    20: (* Transition Delay After Last Bin (Bin 10) Closes *)
        Active_Material_ID := 0;
        Active_Bin_ID := 0;
        Active_Target_Weight := 0.0;
        Status_Message := 'Settling Last Bin';
        Transition_Timer(IN := TRUE, PT := Step_Delay_Time);
        IF Transition_Timer.Q THEN
            Transition_Timer(IN := FALSE);
            Step := 30; // Go to post-discharge wait step (State 30)
        END_IF;

    30: (* Wait 2 Seconds After Closing the Last Bin *)
        Active_Material_ID := 0;
        Active_Bin_ID := 0;
        Active_Target_Weight := 0.0;
        Status_Message := 'Settling Delay';
        Completion_Timer(IN := TRUE, PT := Post_Complete_Delay);
        IF Completion_Timer.Q THEN
            Completion_Timer(IN := FALSE);
            Step := 40; // Proceed to reset last weight (State 40)
        END_IF;
        
    40: (* Reset bin_last_weight to 0 & Complete *)
        Active_Material_ID := 0;
        Active_Bin_ID := 0;
        Active_Target_Weight := 0.0;
        Status_Message := 'Sequence Completed';
        bin_last_weight := 0.0;
        Sequence_Complete := TRUE;
        
        IF NOT Start_Button THEN
            Step := 0;
            Sequence_Complete := FALSE;
            (* Reset all actual weights at completion once start is released *)
            FOR i := 1 TO 10 DO
                Actual_Weights[i] := 0.0;
            END_FOR;
        END_IF;
        
    99: (* Error Abort state *)
        FOR i := 1 TO 10 DO 
            Manual_Bin[i] := FALSE;
            manual_bin_cutoff[i] := FALSE;
            manual_bin_motor[i] := FALSE;
        END_FOR;
        Active_Material_ID := 0;
        Active_Bin_ID := 0;
        Active_Target_Weight := 0.0;
        
        (* Prevent reset loop by checking E_Stop_Active *)
        IF NOT Start_Button AND NOT E_Stop_Active THEN
            Step := 0;
            Error_Code := 0;
            Status_Message := 'Manual Idle';
        END_IF;
END_CASE;

END_FUNCTION_BLOCK

// PLC_AC500_V3/Application/old_version/batching10
PROGRAM batching10
VAR
    Auto_Ctrl : Auto_Batching_V10;
    Manual_Ctrl : Manual_Batching_V10;
    
    (* Global Inputs & Toggles *)
    Start_Button : BOOL;
    E_Stop_Active : BOOL;
    
    (* Parallel Weight Feedbacks *)
    load_cell_auto : REAL;
    load_cell_manual : REAL;
    
    (* Repetitive Cycle Configurations & Status *)
    Target_Batch_Cycles : INT := 2;      // Number of cycles to run automatically (Default: 2)
    Current_Batch_Cycle : INT := 0;      // Current running cycle index
    Completed_Batch_Cycles : INT := 0;  // Total completed batch cycle loops
    All_Cycles_Complete : BOOL;         // Indicator for full set completion
    
    (* Sub-Block Diagnostic Indicators - Ordered exactly below loadcell *)
    Auto_Active_Mat : INT;
    Auto_Active_Bin : INT;
    Auto_Active_Target : REAL; // Active Target Weight for Auto (displays GVL setpoint - Tolerance)
    Auto_Err : INT;
    Auto_Msg : STRING;
    
    Manual_Active_Mat : INT;
    Manual_Active_Bin : INT;
    Manual_Active_Target : REAL; // Active Target Weight for Manual (displays GVL setpoint - Tolerance)
    Manual_Err : INT;
    Manual_Msg : STRING;
    
    (* Process Outputs *)
    Auto_Bin : ARRAY[1..6] OF BOOL; // Valve control outputs (Coarse)
    auto_bin_cutoff : ARRAY[1..6] OF BOOL; // Cutoff indicators (Fine)
    auto_bin_motor : ARRAY[1..6] OF BOOL; // Conveyor/feeder motor outputs
    
    Manual_Bin : ARRAY[1..10] OF BOOL; // Prompt indicators (Coarse)
    manual_bin_cutoff : ARRAY[1..10] OF BOOL; // Cutoff indicators (Fine)
    manual_bin_motor : ARRAY[1..10] OF BOOL; // Conveyor/feeder motor outputs
    
    Auto_Weights : ARRAY[1..6] OF REAL;
    Manual_Weights : ARRAY[1..10] OF REAL;
    
    Auto_Complete : BOOL;
    Manual_Complete : BOOL;
    
    (* Diagnostics & Interlocks *)
    Error_Code : INT := 0;
    Status_Message : STRING := 'System Ready';
    
    (* Array Configurations & Mapping - Renamed for clarity *)
    Auto_Bin_Material_Mapping : ARRAY[1..6] OF INT := [1, 2, 0, 4, 5, 6];
    Manual_Bin_Material_Mapping : ARRAY[1..10] OF INT := [7, 8, 0, 10, 11, 12, 13, 14, 15, 16];
    Auto_Coarse_To_Fine_speed : ARRAY[1..6] OF REAL := [2.0, 1.5, 0.0, 3.0, 5.0, 1.0]; // Cutoff margins (kg)
    Manual_Coarse_To_Fine_speed : ARRAY[1..10] OF REAL := [2.0, 1.5, 0.0, 3.0, 5.0, 1.0, 2.0, 2.0, 2.0, 2.0];
    Auto_Bin_Tolerance : ARRAY[1..6] OF REAL := [1.0, 0.5, 0.0, 1.0, 2.0, 0.5]; // Tolerance offsets (kg)
    Manual_Bin_Tolerance : ARRAY[1..10] OF REAL := [1.0, 0.5, 0.0, 1.0, 2.0, 0.5, 1.0, 1.0, 1.0, 1.0];
    
    i : INT;
    j : INT;
    Duplicate_Found : BOOL;
    Invalid_Material_Range : BOOL;
    
    (* Cycle Manager state variables *)
    Cycle_Manager_State : INT := 0;     // State index for loop management
    Internal_FB_Start : BOOL := FALSE;  // Controlled command to restart sub-blocks
END_VAR

(* 1. STARTUP CONFIGURATION CHECKS *)
Duplicate_Found := FALSE;
Invalid_Material_Range := FALSE;

FOR i := 1 TO 6 DO
    (* Check 2: Out of Range (Auto) *)
    IF Auto_Bin_Material_Mapping[i] < 0 OR Auto_Bin_Material_Mapping[i] > 20 THEN
        Invalid_Material_Range := TRUE;
    END_IF;
    
    (* Check 1: Duplicate Cross-Array Material ID *)
    IF Auto_Bin_Material_Mapping[i] <> 0 AND Auto_Bin_Material_Mapping[i] <= 20 THEN
        FOR j := 1 TO 10 DO
            IF Auto_Bin_Material_Mapping[i] = Manual_Bin_Material_Mapping[j] THEN
                Duplicate_Found := TRUE;
            END_IF;
        END_FOR;
    END_IF;
END_FOR;

FOR j := 1 TO 10 DO
    (* Check 2: Out of Range (Manual) *)
    IF Manual_Bin_Material_Mapping[j] < 0 OR Manual_Bin_Material_Mapping[j] > 20 THEN
        Invalid_Material_Range := TRUE;
    END_IF;
END_FOR;

(* Configuration Error Resolution *)
IF Duplicate_Found THEN
    Error_Code := 1;
    Status_Message := 'Error 1: Duplicate Material ID mapped in Auto and Manual!';
ELSIF Invalid_Material_Range THEN
    Error_Code := 2;
    Status_Message := 'Error 2: Material Index configuration out of range (1..20)!';
ELSE
    IF Error_Code <= 2 THEN
        Error_Code := 0;
    END_IF;
END_IF;

(* Abort sequences if a configuration error exists or E-stop is active *)
IF (Error_Code >= 1 AND Error_Code <= 2) OR E_Stop_Active THEN
    FOR i := 1 TO 6 DO Auto_Bin[i] := FALSE; auto_bin_cutoff[i] := FALSE; auto_bin_motor[i] := FALSE; END_FOR;
    FOR i := 1 TO 10 DO Manual_Bin[i] := FALSE; manual_bin_cutoff[i] := FALSE; manual_bin_motor[i] := FALSE; END_FOR;
    
    Internal_FB_Start := FALSE;
    Auto_Ctrl(Start_Button := FALSE, E_Stop_Active := TRUE, load_cell_value := load_cell_auto);
    Manual_Ctrl(Start_Button := FALSE, E_Stop_Active := TRUE, load_cell_value := load_cell_manual);
    
    Auto_Active_Target := 0.0;
    Manual_Active_Target := 0.0;
    All_Cycles_Complete := FALSE;
    Cycle_Manager_State := 0;
    
    IF E_Stop_Active THEN
        Error_Code := 12;
        Status_Message := 'Error 12: Emergency Stop Active!';
    END_IF;
    RETURN;
END_IF;


(* 2. REPETITIVE CYCLE MANAGER STATE MACHINE *)
CASE Cycle_Manager_State OF
    0: (* IDLE STATE *)
        Internal_FB_Start := FALSE;
        All_Cycles_Complete := FALSE;
        IF Error_Code = 0 THEN Status_Message := 'System Ready'; END_IF;
        
        IF Start_Button THEN
            Current_Batch_Cycle := 1;
            Completed_Batch_Cycles := 0;
            Cycle_Manager_State := 1;
        END_IF;
        
    1: (* RUN STATE (Run Sub-Blocks) *)
        Internal_FB_Start := TRUE;
        Status_Message := CONCAT('Running Batch Cycle ', INT_TO_STRING(Current_Batch_Cycle));
        
        (* Monitor completion of active step *)
        IF Auto_Complete AND Manual_Complete THEN
            Cycle_Manager_State := 2;
        END_IF;
        
    2: (* CHECK REPEAT CYCLE STATE *)
        Completed_Batch_Cycles := Current_Batch_Cycle;
        
        IF Current_Batch_Cycle < Target_Batch_Cycles THEN
            (* Transition to reset pulse to restart FBs *)
            Cycle_Manager_State := 3;
        else
            (* All loop cycles complete *)
            Cycle_Manager_State := 4;
        END_IF;
        
    3: (* AUTO-RESET PULSE (Pulse Start command low to reset state machines) *)
        Internal_FB_Start := FALSE;
        Status_Message := 'Resetting Sequence for Next Cycle';
        
        (* Verify sub-blocks have fully reset to idle step *)
        IF NOT Auto_Complete AND NOT Manual_Complete THEN
            Current_Batch_Cycle := Current_Batch_Cycle + 1;
            Cycle_Manager_State := 1; // Start next cycle
        END_IF;
        
    4: (* SEQUENCE FULLY COMPLETED STATE *)
        Internal_FB_Start := FALSE;
        All_Cycles_Complete := TRUE;
        Status_Message := 'All Batch Cycles Completed';
        
        IF NOT Start_Button THEN
            Cycle_Manager_State := 0;
        END_IF;
END_CASE;


(* 3. CONCURRENT EXECUTION OF FB INSTANCES *)
Auto_Ctrl(
    Start_Button := Internal_FB_Start,
    E_Stop_Active := E_Stop_Active,
    load_cell_value := load_cell_auto,
    Auto_Bin_Material_Mapping := Auto_Bin_Material_Mapping,
    Auto_Coarse_To_Fine_speed := Auto_Coarse_To_Fine_speed,
    Auto_Bin_Tolerance := Auto_Bin_Tolerance,
    Auto_Bin => Auto_Bin,
    auto_bin_cutoff => auto_bin_cutoff,
    auto_bin_motor => auto_bin_motor,
    Actual_Weights => Auto_Weights,
    Sequence_Complete => Auto_Complete,
    Active_Material_ID => Auto_Active_Mat,
    Active_Bin_ID => Auto_Active_Bin,
    Active_Target_Weight => Auto_Active_Target,
    Error_Code => Auto_Err,
    Status_Message => Auto_Msg
);

Manual_Ctrl(
    Start_Button := Internal_FB_Start,
    E_Stop_Active := E_Stop_Active,
    load_cell_value := load_cell_manual,
    Manual_Bin_Material_Mapping := Manual_Bin_Material_Mapping,
    Manual_Coarse_To_Fine_speed := Manual_Coarse_To_Fine_speed,
    Manual_Bin_Tolerance := Manual_Bin_Tolerance,
    Manual_Bin => Manual_Bin,
    manual_bin_cutoff => manual_bin_cutoff,
    manual_bin_motor => manual_bin_motor,
    Actual_Weights => Manual_Weights,
    Sequence_Complete => Manual_Complete,
    Active_Material_ID => Manual_Active_Mat,
    Active_Bin_ID => Manual_Active_Bin,
    Active_Target_Weight => Manual_Active_Target,
    Error_Code => Manual_Err,
    Status_Message => Manual_Msg
);

(* Runtime Error Mapping & Aggregation *)
IF Auto_Err <> 0 THEN
    Error_Code := Auto_Err;
    Status_Message := CONCAT('Auto Error: ', Auto_Msg);
ELSIF Manual_Err <> 0 THEN
    Error_Code := Manual_Err;
    Status_Message := CONCAT('Manual Error: ', Manual_Msg);
ELSIF Cycle_Manager_State = 0 THEN
    Error_Code := 0;
END_IF;

END_PROGRAM

// PLC_AC500_V3/Application/old_version/batching11
PROGRAM batching11
VAR
    Auto_Ctrl : Auto_Batching_V11;
    Semi_Auto_Ctrl : Semi_Auto_Batching_V11;
    
    (* Parallel Weight Feedbacks *)
    load_cell_auto : REAL;
    load_cell_semi_auto : REAL;
    
    (* Sub-Block Diagnostic Indicators (not in GVL) *)
    Auto_Active_Target : REAL; // Active Target Weight for Auto (displays GVL setpoint - Tolerance)
    Auto_Err : INT;
    Auto_Msg : STRING;
    
    Semi_Auto_Active_Target : REAL; // Active Target Weight for Semi-Auto (displays GVL setpoint - Tolerance)
    Semi_Auto_Err : INT;
    Semi_Auto_Msg : STRING;
    
    (* Process Outputs *)
    Auto_Bin : ARRAY[1..6] OF BOOL; // Valve control outputs (Coarse)
    auto_bin_cutoff : ARRAY[1..6] OF BOOL; // Cutoff indicators (Fine)
    auto_bin_motor : ARRAY[1..6] OF BOOL; // Conveyor/feeder motor outputs
    
    Semi_Auto_Bin : ARRAY[1..10] OF BOOL; // Prompt indicators (Coarse)
    semi_auto_bin_cutoff : ARRAY[1..10] OF BOOL; // Cutoff indicators (Fine)
    semi_auto_bin_motor : ARRAY[1..10] OF BOOL; // Conveyor/feeder motor outputs
    
    Auto_Weights : ARRAY[1..6] OF REAL;
    Semi_Auto_Weights : ARRAY[1..10] OF REAL;
    
    Auto_Complete : BOOL;
    Semi_Auto_Complete : BOOL;
    
    (* Repetitive Cycle Status (not in GVL) *)
    Completed_Batch_Cycles : INT := 0;  // Total completed batch cycle loops
    All_Cycles_Complete : BOOL;         // Indicator for full set completion
    
    (* Diagnostics & Interlocks (not in GVL) *)
    Status_Message : STRING := 'System Ready';
    
    i : INT;
    j : INT;
    Duplicate_Found : BOOL;
    Invalid_Material_Range : BOOL;
    
    (* Cycle Manager state variables *)
    Cycle_Manager_State : INT := 0;     // State index for loop management
    Internal_FB_Start : BOOL := FALSE;  // Controlled command to restart sub-blocks
END_VAR

(* 1. STARTUP CONFIGURATION CHECKS *)
Duplicate_Found := FALSE;
Invalid_Material_Range := FALSE;

FOR i := 1 TO 6 DO
    (* Check 2: Out of Range (Auto) *)
    IF GVL.Auto_Bin_Material_Mapping[i] < 0 OR GVL.Auto_Bin_Material_Mapping[i] > 20 THEN
        Invalid_Material_Range := TRUE;
    END_IF;
    
    (* Check 1: Duplicate Cross-Array Material ID *)
    IF GVL.Auto_Bin_Material_Mapping[i] <> 0 AND GVL.Auto_Bin_Material_Mapping[i] <= 20 THEN
        FOR j := 1 TO 10 DO
            IF GVL.Auto_Bin_Material_Mapping[i] = GVL.Semi_Auto_Bin_Material_Mapping[j] THEN
                Duplicate_Found := TRUE;
            END_IF;
        END_FOR;
    END_IF;
END_FOR;

FOR j := 1 TO 10 DO
    (* Check 2: Out of Range (Semi-Auto) *)
    IF GVL.Semi_Auto_Bin_Material_Mapping[j] < 0 OR GVL.Semi_Auto_Bin_Material_Mapping[j] > 20 THEN
        Invalid_Material_Range := TRUE;
    END_IF;
END_FOR;

(* Configuration Error Resolution *)
IF Duplicate_Found THEN
    GVL.Error_Code := 1;
    Status_Message := 'Error 1: Duplicate Material ID mapped in Auto and Semi-Auto!';
ELSIF Invalid_Material_Range THEN
    GVL.Error_Code := 2;
    Status_Message := 'Error 2: Material Index configuration out of range (1..20)!';
ELSE
    IF GVL.Error_Code <= 2 THEN
        GVL.Error_Code := 0;
    END_IF;
END_IF;

(* Abort/Clear arrays if Configuration error is active or Hard Reset is pressed *)
IF (GVL.Error_Code >= 1 AND GVL.Error_Code <= 2) OR GVL.Reset THEN
    FOR i := 1 TO 6 DO Auto_Bin[i] := FALSE; auto_bin_cutoff[i] := FALSE; auto_bin_motor[i] := FALSE; END_FOR;
    FOR i := 1 TO 10 DO Semi_Auto_Bin[i] := FALSE; semi_auto_bin_cutoff[i] := FALSE; semi_auto_bin_motor[i] := FALSE; END_FOR;
    
    Internal_FB_Start := FALSE;
    Auto_Ctrl(Start_Button := FALSE, E_Stop_Active := FALSE, Reset := GVL.Reset, load_cell_value := load_cell_auto);
    Semi_Auto_Ctrl(Start_Button := FALSE, E_Stop_Active := FALSE, Reset := GVL.Reset, load_cell_value := load_cell_semi_auto);
    
    Auto_Active_Target := 0.0;
    Semi_Auto_Active_Target := 0.0;
    All_Cycles_Complete := FALSE;
    GVL.Cycle_Hold_Active := FALSE;
    Cycle_Manager_State := 0;
    
    IF GVL.Reset THEN
        GVL.Error_Code := 0;
        Status_Message := 'System Reset Activated';
    END_IF;
    RETURN;
END_IF;


(* 2. REPETITIVE CYCLE MANAGER STATE MACHINE WITH HOLD RELEASE *)
CASE Cycle_Manager_State OF
    0: (* IDLE STATE *)
        Internal_FB_Start := FALSE;
        All_Cycles_Complete := FALSE;
        GVL.Cycle_Hold_Active := FALSE;
        IF GVL.Error_Code = 0 THEN Status_Message := 'System Ready'; END_IF;
        
        IF GVL.Start_Button THEN
            GVL.Current_Batch_Cycle := 1;
            Completed_Batch_Cycles := 0;
            Cycle_Manager_State := 1;
        END_IF;
        
    1: (* RUN STATE (Run Sub-Blocks) *)
        Internal_FB_Start := TRUE;
        Status_Message := CONCAT('Running Batch Cycle ', INT_TO_STRING(GVL.Current_Batch_Cycle));
        
        (* Monitor completion of active step *)
        IF Auto_Complete AND Semi_Auto_Complete THEN
            Cycle_Manager_State := 2;
        END_IF;
        
    2: (* CHECK REPEAT CYCLE STATE *)
        Completed_Batch_Cycles := GVL.Current_Batch_Cycle;
        
        IF GVL.Current_Batch_Cycle < GVL.Target_Batch_Cycles THEN
            (* Hold cycle loop progression *)
            GVL.Cycle_Hold_Active := TRUE;
            Cycle_Manager_State := 5; // Go to hold wait state
        else
            (* All loop cycles complete *)
            Cycle_Manager_State := 4;
        END_IF;
        
    5: (* PAUSED BETWEEN CYCLES (Holds program until GVL.Cycle_Hold_Active turns FALSE) *)
        Internal_FB_Start := TRUE; // Keep FBs active in finished step state
        Status_Message := CONCAT('Cycle ', CONCAT(INT_TO_STRING(GVL.Current_Batch_Cycle), ' Complete. Waiting to Release.'));
        
        (* Operator toggles hold status back to FALSE to proceed *)
        IF NOT GVL.Cycle_Hold_Active THEN
            Cycle_Manager_State := 3; // Go to auto-reset pulse
        END_IF;
        
    3: (* AUTO-RESET PULSE (Pulse Start command low to reset state machines) *)
        Internal_FB_Start := FALSE;
        Status_Message := 'Resetting Sequence for Next Cycle';
        
        (* Verify sub-blocks have fully reset to idle step *)
        IF NOT Auto_Complete AND NOT Semi_Auto_Complete THEN
            GVL.Current_Batch_Cycle := GVL.Current_Batch_Cycle + 1;
            Cycle_Manager_State := 1; // Start next cycle
        END_IF;
        
    4: (* SEQUENCE FULLY COMPLETED STATE *)
        Internal_FB_Start := FALSE;
        All_Cycles_Complete := TRUE;
        Status_Message := 'All Batch Cycles Completed';
        
        IF NOT GVL.Start_Button THEN
            Cycle_Manager_State := 0;
        END_IF;
END_CASE;


(* 3. CONCURRENT EXECUTION OF FB INSTANCES *)
Auto_Ctrl(
    Start_Button := Internal_FB_Start,
    E_Stop_Active := GVL.E_Stop_Active,
    Reset := GVL.Reset,
    load_cell_value := load_cell_auto,
    Auto_Bin_Material_Mapping := GVL.Auto_Bin_Material_Mapping,
    Auto_Coarse_To_Fine_speed := GVL.Auto_Coarse_To_Fine_speed,
    Auto_Bin_Tolerance := GVL.Auto_Bin_Tolerance,
    Auto_Bin => Auto_Bin,
    auto_bin_cutoff => auto_bin_cutoff,
    auto_bin_motor => auto_bin_motor,
    Actual_Weights => Auto_Weights,
    Sequence_Complete => Auto_Complete,
    Active_Material_ID => GVL.Auto_Active_Mat,
    Active_Bin_ID => GVL.Auto_Active_Bin,
    Active_Target_Weight => Auto_Active_Target,
    Error_Code => Auto_Err,
    Status_Message => Auto_Msg
);

Semi_Auto_Ctrl(
    Start_Button := Internal_FB_Start,
    E_Stop_Active := GVL.E_Stop_Active,
    Reset := GVL.Reset,
    load_cell_value := load_cell_semi_auto,
    Semi_Auto_Bin_Material_Mapping := GVL.Semi_Auto_Bin_Material_Mapping,
    Semi_Auto_Coarse_To_Fine_speed := GVL.Semi_Auto_Coarse_To_Fine_speed,
    Semi_Auto_Bin_Tolerance := GVL.Semi_Auto_Bin_Tolerance,
    Semi_Auto_Bin => Semi_Auto_Bin,
    semi_auto_bin_cutoff => semi_auto_bin_cutoff,
    semi_auto_bin_motor => semi_auto_bin_motor,
    Actual_Weights => Semi_Auto_Weights,
    Sequence_Complete => Semi_Auto_Complete,
    Active_Material_ID => GVL.Semi_Auto_Active_Mat,
    Active_Bin_ID => GVL.Semi_Auto_Active_Bin,
    Active_Target_Weight => Semi_Auto_Active_Target,
    Error_Code => Semi_Auto_Err,
    Status_Message => Semi_Auto_Msg
);

(* Runtime Error Mapping & Aggregation *)
IF Auto_Err <> 0 THEN
    GVL.Error_Code := Auto_Err;
    Status_Message := CONCAT('Auto Error: ', Auto_Msg);
ELSIF Semi_Auto_Err <> 0 THEN
    GVL.Error_Code := Semi_Auto_Err;
    Status_Message := CONCAT('Semi-Auto Error: ', Semi_Auto_Msg);
ELSIF Cycle_Manager_State = 0 THEN
    GVL.Error_Code := 0;
END_IF;

END_PROGRAM

// PLC_AC500_V3/Application/old_version/Auto_Batching_V11
FUNCTION_BLOCK Auto_Batching_V11
VAR_INPUT
    Start_Button : BOOL;      // Signal to start/resume the batching sequence
    E_Stop_Active : BOOL;     // Emergency Stop (Pause/Hold signal)
    Reset : BOOL;             // Hard reset sequence back to idle state
    Auto_Bin_Material_Mapping : ARRAY[1..6] OF INT; // Material index mapping for 6 bins
    Auto_Coarse_To_Fine_speed : ARRAY[1..6] OF REAL; // Cutoff weight thresholds (kg)
    Auto_Bin_Tolerance : ARRAY[1..6] OF REAL; // Tolerance weight offset values (kg)
END_VAR
VAR_IN_OUT
    load_cell_value : REAL;   // Weight value read/written from load cell
END_VAR
VAR_OUTPUT
    Auto_Bin : ARRAY[1..6] OF BOOL; // Coarse feed valve outputs
    auto_bin_cutoff : ARRAY[1..6] OF BOOL; // Fine feed cutoff trigger indicators
    auto_bin_motor : ARRAY[1..6] OF BOOL; // Main conveyor motor outputs
    Actual_Weights : ARRAY[1..6] OF REAL; // Actual weight poured per silo
    Sequence_Complete : BOOL;  // Batch complete flag
    Active_Material_ID : INT;  // Currently active ingredient ID
    Active_Bin_ID : INT;       // Currently active physical Bin ID (1..6)
    Active_Target_Weight : REAL; // Recipe target weight of active bin (with tolerance applied)
    Error_Code : INT;          // Active error code
    Status_Message : STRING;   // Diagnostic text message
END_VAR
VAR
    Step : INT := 0;          // State machine index (0: Idle, 1..6: Bins, 11..16: Delays, 7: Settling, 8: Complete)
    bin_last_weight : REAL;   // Baseline weight snapshot before starting current bin
    actual_bin : REAL;        // Current weight added from active bin
    target_act_bin : REAL;    // Effective target weight to add from the active bin (GVL target - Tolerance)
    cutoff_trigger_weight : REAL; // Calculated trigger weight (target - Tolerance - Cutoff)
    Paused_By_EStop : BOOL := FALSE; // Pause status latch
    
    Mat_Idx : INT;
    i : INT;                  // General loop index
    
    (* TIMERS FOR TRANSITIONS & DELAYS *)
    Transition_Timer : TON;
    Completion_Timer : TON;
    Step_Delay_Time : TIME := T#2S;
    Post_Complete_Delay : TIME := T#2S;
    
    (* SELF-CONTAINED SIMULATION VARIABLES *)
    Simulation_Mode : BOOL := TRUE;
    Sim_Rate : REAL := 10.0;            // Simulated pouring speed (10.0 kg/s)
    Sim_Timer : TON;
    Start_Sim_Weight : REAL;
    Discharge_Active : BOOL;
END_VAR

(* Auto Batching FB V11 with E-Stop Pause & Reset Logic *)

(* 1. HARD RESET INTERLOCK (Resets weights immediately) *)
IF Reset THEN
    FOR i := 1 TO 6 DO
        Auto_Bin[i] := FALSE;
        auto_bin_cutoff[i] := FALSE;
        auto_bin_motor[i] := FALSE;
        Actual_Weights[i] := 0.0;
    END_FOR;
    Sequence_Complete := FALSE;
    Active_Material_ID := 0;
    Active_Bin_ID := 0;
    Active_Target_Weight := 0.0;
    Error_Code := 0;
    Status_Message := 'Auto Reset Activated';
    Paused_By_EStop := FALSE;
    Step := 0;
    
    (* Clear simulation weights immediately *)
    load_cell_value := 0.0;
    bin_last_weight := 0.0;
    Start_Sim_Weight := 0.0;
    
    Transition_Timer(IN := FALSE);
    Completion_Timer(IN := FALSE);
    Sim_Timer(IN := FALSE);
    RETURN;
END_IF;

(* 2. E-STOP PAUSE / HOLD LOGIC *)
IF E_Stop_Active THEN
    Paused_By_EStop := TRUE;
END_IF;

IF Paused_By_EStop THEN
    (* Suspend all valve/motor control outputs immediately *)
    FOR i := 1 TO 6 DO
        Auto_Bin[i] := FALSE;
        auto_bin_cutoff[i] := FALSE;
        auto_bin_motor[i] := FALSE;
    END_FOR;
    
    IF E_Stop_Active THEN
        Status_Message := 'Auto Paused: Emergency Stop Active!';
    ELSE
        Status_Message := 'Auto Paused: Press Start to Resume';
        
        (* Resume sequence when Start Button is pressed *)
        IF Start_Button THEN
            Paused_By_EStop := FALSE;
        END_IF;
    END_IF;
    
    (* Freeze simulation timers and exit code execution (Hold current Step) *)
    Sim_Timer(IN := FALSE);
    Transition_Timer(IN := FALSE);
    Completion_Timer(IN := FALSE);
    RETURN;
END_IF;

(* 3. SELF-CONTAINED SIMULATION WEIGHT MANAGEMENT *)
IF Simulation_Mode THEN
    (* Reset simulation to baseline *)
    IF Step = 0 AND NOT Start_Button AND NOT Sequence_Complete THEN
        load_cell_value := 0.0;
        bin_last_weight := 0.0;
        Start_Sim_Weight := 0.0;
        Sim_Timer(IN := FALSE);
    END_IF;
    
    (* Check if any valve is actively discharging *)
    Discharge_Active := FALSE;
    IF Step >= 1 AND Step <= 6 THEN
        Discharge_Active := auto_bin_motor[Step];
    END_IF;
    
    (* Simulate weight gain on the load cell *)
    IF Discharge_Active THEN
        Sim_Timer(IN := TRUE, PT := T#1000S);
        load_cell_value := Start_Sim_Weight + (TIME_TO_REAL(Sim_Timer.ET) / 1000.0) * Sim_Rate;
    ELSE
        Sim_Timer(IN := FALSE);
        Start_Sim_Weight := load_cell_value;
    END_IF;
END_IF;


(* 4. RECIPE SEQUENCE START *)
IF Step = 0 AND Start_Button THEN
    Step := 1;
    bin_last_weight := load_cell_value;
    Sequence_Complete := FALSE;
    Error_Code := 0;
    Status_Message := 'Auto Pour Started';
    Active_Target_Weight := 0.0;
    (* Clear actual weights and outputs on start *)
    FOR i := 1 TO 6 DO
        Actual_Weights[i] := 0.0;
        Auto_Bin[i] := FALSE;
        auto_bin_cutoff[i] := FALSE;
        auto_bin_motor[i] := FALSE;
    END_FOR;
END_IF;


(* 5. SEQUENCE CONTROL STATE MACHINE *)
CASE Step OF
    0:
        Active_Material_ID := 0;
        Active_Bin_ID := 0;
        Active_Target_Weight := 0.0;
        IF Error_Code = 0 THEN Status_Message := 'Auto Idle'; END_IF;
        
    1..6: (* Discharging Silos 1 to 6 *)
        Mat_Idx := Auto_Bin_Material_Mapping[Step];
        
        (* Skip this step instantly if material mapping is 0 OR target weight is 0.0 kg *)
        IF Mat_Idx = 0 OR (Mat_Idx <= 20 AND GVL.Recipe_Weights[Mat_Idx] = 0.0) THEN
            Step := Step + 1;
        ELSE
            (* Calculate effective target weight (Looked up Target - Tolerance) *)
            target_act_bin := GVL.Recipe_Weights[Mat_Idx] - Auto_Bin_Tolerance[Step];
            Active_Target_Weight := target_act_bin;
            
            (* Calculate weight added by current active bin *)
            actual_bin := load_cell_value - bin_last_weight;
            Actual_Weights[Step] := actual_bin;
            
            (* Calculate cutoff trigger threshold *)
            cutoff_trigger_weight := target_act_bin - Auto_Coarse_To_Fine_speed[Step];
            
            Active_Material_ID := Mat_Idx;
            Active_Bin_ID := Step;
            Status_Message := 'Auto Pouring';
            
            (* COARSE/FINE FEED TRANSITIONS WITH TOLERANCE OFFSETS *)
            IF actual_bin < cutoff_trigger_weight THEN
                (* Phase 1: Coarse Feed *)
                Auto_Bin[Step] := TRUE;
                auto_bin_cutoff[Step] := FALSE;
                auto_bin_motor[Step] := TRUE;
            ELSIF actual_bin < target_act_bin THEN
                (* Phase 2: Fine Feed *)
                Auto_Bin[Step] := FALSE;
                auto_bin_cutoff[Step] := TRUE;
                auto_bin_motor[Step] := TRUE;
            ELSE
                (* Phase 3: Completed (All OFF) *)
                Auto_Bin[Step] := FALSE;
                auto_bin_cutoff[Step] := FALSE;
                auto_bin_motor[Step] := FALSE;
                bin_last_weight := load_cell_value;
                Active_Target_Weight := 0.0;
                Step := 10 + Step; // Offset to separate transition states
            END_IF;
            
            (* RUNTIME CHECKS *)
            (* Check 21 & 22: Scale Limits *)
            IF load_cell_value > 500.0 THEN
                Error_Code := 21;
                Status_Message := 'Error 21: Scale Overloaded!';
                Paused_By_EStop := TRUE; // Pause sequence on fault
            ELSIF load_cell_value < 0.0 THEN
                Error_Code := 22;
                Status_Message := 'Error 22: Scale Underloaded/Fault!';
                Paused_By_EStop := TRUE; // Pause sequence on fault
            END_IF;
        END_IF;

    11..15: (* Transition Delays (Between Bins) *)
        Active_Material_ID := 0;
        Active_Bin_ID := 0;
        Active_Target_Weight := 0.0;
        Status_Message := 'Transition Delay';
        
        Transition_Timer(IN := TRUE, PT := Step_Delay_Time);
        IF Transition_Timer.Q THEN
            Transition_Timer(IN := FALSE);
            Step := (Step - 10) + 1; // Advance to next bin
        END_IF;
        
    16: (* Transition Delay After Last Bin (Bin 6) Closes *)
        Active_Material_ID := 0;
        Active_Bin_ID := 0;
        Active_Target_Weight := 0.0;
        Status_Message := 'Settling Last Bin';
        
        Transition_Timer(IN := TRUE, PT := Step_Delay_Time);
        IF Transition_Timer.Q THEN
            Transition_Timer(IN := FALSE);
            Step := 7; // Go to post-discharge wait step
        END_IF;

    7: (* Wait 2 Seconds After Closing the Last Bin *)
        Active_Material_ID := 0;
        Active_Bin_ID := 0;
        Active_Target_Weight := 0.0;
        Status_Message := 'Settling Delay';
        Completion_Timer(IN := TRUE, PT := Post_Complete_Delay);
        IF Completion_Timer.Q THEN
            Completion_Timer(IN := FALSE);
            Step := 8; // Proceed to reset last weight
        END_IF;
        
    8: (* Reset bin_last_weight to 0 & Complete *)
        Active_Material_ID := 0;
        Active_Bin_ID := 0;
        Active_Target_Weight := 0.0;
        Status_Message := 'Sequence Completed';
        bin_last_weight := 0.0;
        Sequence_Complete := TRUE;
        
        IF NOT Start_Button THEN
            Step := 0;
            Sequence_Complete := FALSE;
            (* Reset all actual weights at completion once start is released *)
            FOR i := 1 TO 6 DO
                Actual_Weights[i] := 0.0;
            END_FOR;
        END_IF;
END_CASE;

END_FUNCTION_BLOCK

// PLC_AC500_V3/Application/old_version/Semi_Auto_Batching_V11
FUNCTION_BLOCK Semi_Auto_Batching_V11
VAR_INPUT
    Start_Button : BOOL;      // Signal to start/resume the batching sequence
    E_Stop_Active : BOOL;     // Emergency Stop (Pause/Hold signal)
    Reset : BOOL;             // Hard reset sequence back to idle state
    Semi_Auto_Bin_Material_Mapping : ARRAY[1..10] OF INT; // Material index mapping for 10 manual silos
    Semi_Auto_Coarse_To_Fine_speed : ARRAY[1..10] OF REAL; // Cutoff weight thresholds (kg)
    Semi_Auto_Bin_Tolerance : ARRAY[1..10] OF REAL; // Tolerance weight offset values (kg)
END_VAR
VAR_IN_OUT
    load_cell_value : REAL;   // Weight value read/written from load cell
END_VAR
VAR_OUTPUT
    Semi_Auto_Bin : ARRAY[1..10] OF BOOL; // Prompts/indicators for Bins 7..16
    semi_auto_bin_cutoff : ARRAY[1..10] OF BOOL; // Manual pre-cutoff indicators
    semi_auto_bin_motor : ARRAY[1..10] OF BOOL; // Main manual feeder motor outputs
    Actual_Weights : ARRAY[1..10] OF REAL; // Actual weight poured per silo
    Sequence_Complete : BOOL;  // Batch complete flag
    Active_Material_ID : INT;  // Currently active ingredient ID
    Active_Bin_ID : INT;       // Currently active physical Bin ID (7..16)
    Active_Target_Weight : REAL; // Recipe target weight of active bin (with tolerance applied)
    Error_Code : INT;          // Active error code
    Status_Message : STRING;   // Diagnostic text message
END_VAR
VAR
    Step : INT := 0;          // State machine index (0: Idle, 1..10: Bins, 11..20: Delays, 30: Settling, 40: Complete)
    bin_last_weight : REAL;   // Baseline weight snapshot before starting current bin
    actual_bin : REAL;        // Current weight added from active bin
    target_act_bin : REAL;    // Effective target weight to add from the active bin (GVL target - Tolerance)
    cutoff_trigger_weight : REAL; // Calculated target threshold weight minus cutoff and tolerance values
    Paused_By_EStop : BOOL := FALSE; // Pause status latch
    
    Mat_Idx : INT;
    i : INT;                  // General loop index
    
    (* TIMERS FOR TRANSITIONS & DELAYS *)
    Transition_Timer : TON;
    Completion_Timer : TON;
    Operator_Timer : TON;
    Step_Delay_Time : TIME := T#2S;
    Post_Complete_Delay : TIME := T#2S;
    
    (* SELF-CONTAINED SIMULATION VARIABLES *)
    Simulation_Mode : BOOL := TRUE;
    Sim_Rate : REAL := 10.0;            // Simulated pouring speed (10.0 kg/s)
    Sim_Timer : TON;
    Start_Sim_Weight : REAL;
    Discharge_Active : BOOL;
END_VAR

(* Semi-Auto Batching FB V11 with E-Stop Pause & Reset Logic *)

(* 1. HARD RESET INTERLOCK (Resets weights immediately) *)
IF Reset THEN
    FOR i := 1 TO 10 DO
        Semi_Auto_Bin[i] := FALSE;
        semi_auto_bin_cutoff[i] := FALSE;
        semi_auto_bin_motor[i] := FALSE;
        Actual_Weights[i] := 0.0;
    END_FOR;
    Sequence_Complete := FALSE;
    Active_Material_ID := 0;
    Active_Bin_ID := 0;
    Active_Target_Weight := 0.0;
    Error_Code := 0;
    Status_Message := 'Semi-Auto Reset Activated';
    Paused_By_EStop := FALSE;
    Step := 0;
    
    (* Clear simulation weights immediately *)
    load_cell_value := 0.0;
    bin_last_weight := 0.0;
    Start_Sim_Weight := 0.0;
    
    Transition_Timer(IN := FALSE);
    Completion_Timer(IN := FALSE);
    Operator_Timer(IN := FALSE);
    Sim_Timer(IN := FALSE);
    RETURN;
END_IF;

(* 2. E-STOP PAUSE / HOLD LOGIC *)
IF E_Stop_Active THEN
    Paused_By_EStop := TRUE;
END_IF;

IF Paused_By_EStop THEN
    (* Suspend all indicators and feeder outputs *)
    FOR i := 1 TO 10 DO
        Semi_Auto_Bin[i] := FALSE;
        semi_auto_bin_cutoff[i] := FALSE;
        semi_auto_bin_motor[i] := FALSE;
    END_FOR;
    
    IF E_Stop_Active THEN
        Status_Message := 'Semi-Auto Paused: Emergency Stop Active!';
    ELSE
        Status_Message := 'Semi-Auto Paused: Press Start to Resume';
        
        (* Resume sequence when Start Button is pressed *)
        IF Start_Button THEN
            Paused_By_EStop := FALSE;
        END_IF;
    END_IF;
    
    (* Freeze simulation and safety timers *)
    Sim_Timer(IN := FALSE);
    Transition_Timer(IN := FALSE);
    Completion_Timer(IN := FALSE);
    Operator_Timer(IN := FALSE);
    RETURN;
END_IF;

(* 3. SELF-CONTAINED SIMULATION WEIGHT MANAGEMENT *)
IF Simulation_Mode THEN
    (* Reset simulation to baseline *)
    IF Step = 0 AND NOT Start_Button AND NOT Sequence_Complete THEN
        load_cell_value := 0.0;
        bin_last_weight := 0.0;
        Start_Sim_Weight := 0.0;
        Sim_Timer(IN := FALSE);
    END_IF;
    
    (* Check if operator is actively pouring *)
    Discharge_Active := FALSE;
    IF Step >= 1 AND Step <= 10 THEN
        Discharge_Active := semi_auto_bin_motor[Step];
    END_IF;
    
    (* Simulate weight gain on the load cell *)
    IF Discharge_Active THEN
        Sim_Timer(IN := TRUE, PT := T#1000S);
        load_cell_value := Start_Sim_Weight + (TIME_TO_REAL(Sim_Timer.ET) / 1000.0) * Sim_Rate;
    ELSE
        Sim_Timer(IN := FALSE);
        Start_Sim_Weight := load_cell_value;
    END_IF;
END_IF;


(* 4. RECIPE SEQUENCE START *)
IF Step = 0 AND Start_Button THEN
    Step := 1;
    bin_last_weight := load_cell_value;
    Sequence_Complete := FALSE;
    Error_Code := 0;
    Status_Message := 'Semi-Auto Pour Started';
    Active_Target_Weight := 0.0;
    (* Clear actual weights on start *)
    FOR i := 1 TO 10 DO
        Actual_Weights[i] := 0.0;
        Semi_Auto_Bin[i] := FALSE;
        semi_auto_bin_cutoff[i] := FALSE;
        semi_auto_bin_motor[i] := FALSE;
    END_FOR;
END_IF;


(* 5. SEQUENCE CONTROL STATE MACHINE *)
CASE Step OF
    0:
        Active_Material_ID := 0;
        Active_Bin_ID := 0;
        Active_Target_Weight := 0.0;
        IF Error_Code = 0 THEN Status_Message := 'Semi-Auto Idle'; END_IF;
        
    1..10: (* Prompts Silos 7 to 16 *)
        Mat_Idx := Semi_Auto_Bin_Material_Mapping[Step];
        
        (* Skip this step instantly if material mapping is 0 OR target weight is 0.0 kg *)
        IF Mat_Idx = 0 OR (Mat_Idx <= 20 AND GVL.Recipe_Weights[Mat_Idx] = 0.0) THEN
            Step := Step + 1;
        ELSE
            (* Calculate effective target weight (Looked up Target - Tolerance) *)
            target_act_bin := GVL.Recipe_Weights[Mat_Idx] - Semi_Auto_Bin_Tolerance[Step];
            Active_Target_Weight := target_act_bin;
            
            (* Calculate weight added by current active bin *)
            actual_bin := load_cell_value - bin_last_weight;
            Actual_Weights[Step] := actual_bin;
            
            (* Calculate cutoff trigger threshold *)
            cutoff_trigger_weight := target_act_bin - Semi_Auto_Coarse_To_Fine_speed[Step];
            
            Active_Material_ID := Mat_Idx;
            Active_Bin_ID := Step;
            Status_Message := 'Semi-Auto Pouring Active';
            
            (* COARSE/FINE FEED TRANSITIONS WITH TOLERANCE OFFSETS *)
            IF actual_bin < cutoff_trigger_weight THEN
                (* Phase 1: Coarse Feed *)
                Semi_Auto_Bin[Step] := TRUE;
                semi_auto_bin_cutoff[Step] := FALSE;
                semi_auto_bin_motor[Step] := TRUE;
            ELSIF actual_bin < target_act_bin THEN
                (* Phase 2: Fine Feed *)
                Semi_Auto_Bin[Step] := FALSE;
                semi_auto_bin_cutoff[Step] := TRUE;
                semi_auto_bin_motor[Step] := TRUE;
            ELSE
                (* Phase 3: Completed (All OFF) *)
                Semi_Auto_Bin[Step] := FALSE;
                semi_auto_bin_cutoff[Step] := FALSE;
                semi_auto_bin_motor[Step] := FALSE;
                bin_last_weight := load_cell_value;
                Active_Target_Weight := 0.0;
                Step := 10 + Step; // Offset to separate transition states
            END_IF;
            
            (* RUNTIME CHECKS *)
            (* Check 21 & 22: Scale Limits *)
            IF load_cell_value > 500.0 THEN
                Error_Code := 21;
                Status_Message := 'Error 21: Scale Overloaded!';
                Paused_By_EStop := TRUE;
            ELSIF load_cell_value < 0.0 THEN
                Error_Code := 22;
                Status_Message := 'Error 22: Scale Underloaded/Fault!';
                Paused_By_EStop := TRUE;
            END_IF;
            
            (* Check 30: Operator Timeout *)
            Operator_Timer(IN := semi_auto_bin_motor[Step], PT := T#300S);
            IF Operator_Timer.Q THEN
                Error_Code := 30;
                Status_Message := 'Error 30: Semi-Auto Operator Timeout!';
                Paused_By_EStop := TRUE;
            END_IF;
        END_IF;

    11..19: (* Transition Delays (Between Bins) *)
        Active_Material_ID := 0;
        Active_Bin_ID := 0;
        Active_Target_Weight := 0.0;
        Status_Message := 'Transition Delay';
        Transition_Timer(IN := TRUE, PT := Step_Delay_Time);
        IF Transition_Timer.Q THEN
            Transition_Timer(IN := FALSE);
            Step := (Step - 10) + 1; // Advance to next bin
        END_IF;
        
    20: (* Transition Delay After Last Bin (Bin 10) Closes *)
        Active_Material_ID := 0;
        Active_Bin_ID := 0;
        Active_Target_Weight := 0.0;
        Status_Message := 'Settling Last Bin';
        Transition_Timer(IN := TRUE, PT := Step_Delay_Time);
        IF Transition_Timer.Q THEN
            Transition_Timer(IN := FALSE);
            Step := 30; // Go to post-discharge wait step (State 30)
        END_IF;

    30: (* Wait 2 Seconds After Closing the Last Bin *)
        Active_Material_ID := 0;
        Active_Bin_ID := 0;
        Active_Target_Weight := 0.0;
        Status_Message := 'Settling Delay';
        Completion_Timer(IN := TRUE, PT := Post_Complete_Delay);
        IF Completion_Timer.Q THEN
            Completion_Timer(IN := FALSE);
            Step := 40; // Proceed to reset last weight (State 40)
        END_IF;
        
    40: (* Reset bin_last_weight to 0 & Complete *)
        Active_Material_ID := 0;
        Active_Bin_ID := 0;
        Active_Target_Weight := 0.0;
        Status_Message := 'Sequence Completed';
        bin_last_weight := 0.0;
        Sequence_Complete := TRUE;
        
        IF NOT Start_Button THEN
            Step := 0;
            Sequence_Complete := FALSE;
            (* Reset all actual weights at completion once start is released *)
            FOR i := 1 TO 10 DO
                Actual_Weights[i] := 0.0;
            END_FOR;
        END_IF;
END_CASE;

END_FUNCTION_BLOCK

// PLC_AC500_V3/Application/old_version/Auto_Batching_V12
FUNCTION_BLOCK Auto_Batching_V12
VAR_INPUT
    Start_Button : BOOL;      // Signal to start/resume the batching sequence
    E_Stop_Active : BOOL;     // Emergency Stop (Pause/Hold signal)
    Reset : BOOL;             // Hard reset sequence back to idle state
    Auto_Bin_Material_Mapping : ARRAY[1..6] OF INT; // Material index mapping for 6 bins
    Auto_Coarse_To_Fine_speed : ARRAY[1..6] OF REAL; // Cutoff weight thresholds (kg)
    Auto_Bin_Tolerance : ARRAY[1..6] OF REAL; // Tolerance weight offset values (kg)
END_VAR
VAR_IN_OUT
    load_cell_value : REAL;   // Weight value read/written from load cell
END_VAR
VAR_OUTPUT
    Auto_Bin : ARRAY[1..6] OF BOOL; // Coarse feed valve outputs
    auto_bin_cutoff : ARRAY[1..6] OF BOOL; // Fine feed cutoff trigger indicators
    auto_bin_motor : ARRAY[1..6] OF BOOL; // Main conveyor motor outputs
    Actual_Weights : ARRAY[1..6] OF REAL; // Actual weight poured per silo
    Sequence_Complete : BOOL;  // Batch complete flag
    Active_Material_ID : INT;  // Currently active ingredient ID
    Active_Bin_ID : INT;       // Currently active physical Bin ID (1..6)
    Active_Target_Weight : REAL; // Recipe target weight of active bin (with tolerance applied)
    Error_Code : INT;          // Active error code
    Status_Message : STRING;   // Diagnostic text message
END_VAR
VAR
    Step : INT;                // State machine index
    bin_last_weight : REAL;   // Baseline weight snapshot before starting current bin
    actual_bin : REAL;        // Current weight added from active bin
    target_act_bin : REAL;    // Effective target weight to add from the active bin
    cutoff_trigger_weight : REAL; // Calculated trigger weight
    Paused_By_EStop : BOOL;    // Pause status latch
    
    Mat_Idx : INT;
    i : INT;                  // General loop index
    
    (* TIMERS FOR TRANSITIONS & DELAYS *)
    Transition_Timer : TON;
    Completion_Timer : TON;
    
    (* SELF-CONTAINED SIMULATION VARIABLES *)
    Simulation_Mode : BOOL;    // Simulation disabled
    Sim_Rate : REAL;
    Sim_Timer : TON;
    Start_Sim_Weight : REAL;
    Discharge_Active : BOOL;
END_VAR

(* Auto Batching FB V12 with E-Stop Pause & Reset Logic *)

(* 1. HARD RESET INTERLOCK (Resets weights immediately) *)
IF Reset THEN
    FOR i := 1 TO 6 DO
        Auto_Bin[i] := FALSE;
        auto_bin_cutoff[i] := FALSE;
        auto_bin_motor[i] := FALSE;
        Actual_Weights[i] := 0.0;
    END_FOR;
    Sequence_Complete := FALSE;
    Active_Material_ID := 0;
    Active_Bin_ID := 0;
    Active_Target_Weight := 0.0;
    Error_Code := 0;
    Status_Message := '';
    Paused_By_EStop := FALSE;
    Step := 0;
    
    load_cell_value := 0.0;
    bin_last_weight := 0.0;
    Start_Sim_Weight := 0.0;
    
    Transition_Timer(IN := FALSE);
    Completion_Timer(IN := FALSE);
    Sim_Timer(IN := FALSE);
    RETURN;
END_IF;

(* 2. E-STOP PAUSE / HOLD LOGIC *)
IF E_Stop_Active THEN
    Paused_By_EStop := TRUE;
END_IF;

IF Paused_By_EStop THEN
    (* Suspend all valve/motor control outputs immediately *)
    FOR i := 1 TO 6 DO
        Auto_Bin[i] := FALSE;
        auto_bin_cutoff[i] := FALSE;
        auto_bin_motor[i] := FALSE;
    END_FOR;
    
    IF E_Stop_Active THEN
        Status_Message := 'Auto Paused: Emergency Stop Active!';
    ELSE
        Status_Message := 'Auto Paused: Press Start to Resume';
        
        (* Resume sequence when Start Button is pressed *)
        IF Start_Button THEN
            Paused_By_EStop := FALSE;
        END_IF;
    END_IF;
    
    (* Freeze simulation timers and exit code execution *)
    Sim_Timer(IN := FALSE);
    Transition_Timer(IN := FALSE);
    Completion_Timer(IN := FALSE);
    RETURN;
END_IF;

(* 3. SELF-CONTAINED SIMULATION WEIGHT MANAGEMENT *)
IF Simulation_Mode THEN
    (* Reset simulation to baseline *)
    IF Step = 0 AND NOT Start_Button AND NOT Sequence_Complete THEN
        load_cell_value := 0.0;
        bin_last_weight := 0.0;
        Start_Sim_Weight := 0.0;
        Sim_Timer(IN := FALSE);
    END_IF;
    
    (* Check if any valve is actively discharging *)
    Discharge_Active := FALSE;
    IF Step >= 1 AND Step <= 6 THEN
        Discharge_Active := auto_bin_motor[Step];
    END_IF;
    
    (* Simulate weight gain on the load cell *)
    IF Discharge_Active THEN
        Sim_Timer(IN := TRUE, PT := T#1000S);
        load_cell_value := Start_Sim_Weight + (TIME_TO_REAL(Sim_Timer.ET) / 1000.0) * Sim_Rate;
    ELSE
        Sim_Timer(IN := FALSE);
        Start_Sim_Weight := load_cell_value;
    END_IF;
END_IF;


(* 4. RECIPE SEQUENCE START *)
IF Step = 0 AND Start_Button THEN
    Step := 1;
    bin_last_weight := load_cell_value;
    Sequence_Complete := FALSE;
    Error_Code := 0;
    Status_Message := 'Auto Pour Started';
    Active_Target_Weight := 0.0;
    (* Clear actual weights and outputs on start *)
    FOR i := 1 TO 6 DO
        Actual_Weights[i] := 0.0;
        Auto_Bin[i] := FALSE;
        auto_bin_cutoff[i] := FALSE;
        auto_bin_motor[i] := FALSE;
    END_FOR;
END_IF;


(* 5. SEQUENCE CONTROL STATE MACHINE *)
CASE Step OF
    0:
        Active_Material_ID := 0;
        Active_Bin_ID := 0;
        Active_Target_Weight := 0.0;
        IF Error_Code = 0 THEN Status_Message := 'Auto Idle'; END_IF;
        
    1..6: (* Discharging Silos 1 to 6 *)
        Mat_Idx := Auto_Bin_Material_Mapping[Step];
        
        (* Skip this step instantly if material mapping is 0 OR target weight is 0.0 kg *)
        IF Mat_Idx = 0 OR (Mat_Idx <= 20 AND GVL.Recipe_Weights[Mat_Idx] = 0.0) THEN
            Step := Step + 1;
        ELSE
            (* Calculate effective target weight (Looked up Target - Tolerance) *)
            target_act_bin := GVL.Recipe_Weights[Mat_Idx] - Auto_Bin_Tolerance[Step];
            Active_Target_Weight := target_act_bin;
            
            (* Calculate weight added by current active bin *)
            actual_bin := load_cell_value - bin_last_weight;
            Actual_Weights[Step] := actual_bin;
            
            (* Calculate cutoff trigger threshold *)
            cutoff_trigger_weight := target_act_bin - Auto_Coarse_To_Fine_speed[Step];
            
            Active_Material_ID := Mat_Idx;
            Active_Bin_ID := Step;
            Status_Message := 'Auto Pouring';
            
            (* COARSE/FINE FEED TRANSITIONS WITH TOLERANCE OFFSETS *)
            IF actual_bin < cutoff_trigger_weight THEN
                (* Phase 1: Coarse Feed *)
                Auto_Bin[Step] := TRUE;
                auto_bin_cutoff[Step] := FALSE;
                auto_bin_motor[Step] := TRUE;
            ELSIF actual_bin < target_act_bin THEN
                (* Phase 2: Fine Feed *)
                Auto_Bin[Step] := FALSE;
                auto_bin_cutoff[Step] := TRUE;
                auto_bin_motor[Step] := TRUE;
            ELSE
                (* Phase 3: Completed (All OFF) *)
                Auto_Bin[Step] := FALSE;
                auto_bin_cutoff[Step] := FALSE;
                auto_bin_motor[Step] := FALSE;
                bin_last_weight := load_cell_value;
                Active_Target_Weight := 0.0;
                Step := 10 + Step; // Offset to separate transition states
            END_IF;
            
            (* RUNTIME CHECKS *)
            (* Check 21 & 22: Scale Limits *)
            IF load_cell_value > 500.0 THEN
                Error_Code := 21;
                Status_Message := 'Error 21: Scale Overloaded!';
                Sequence_Complete := TRUE; // Mark complete on halt
                Paused_By_EStop := TRUE; // Pause sequence on fault
            ELSIF load_cell_value < 0.0 THEN
                Error_Code := 22;
                Status_Message := 'Error 22: Scale Underloaded/Fault!';
                Sequence_Complete := TRUE; // Mark complete on halt
                Paused_By_EStop := TRUE; // Pause sequence on fault
            END_IF;
        END_IF;

    11..15: (* Transition Delays (Between Bins) *)
        Active_Material_ID := 0;
        Active_Bin_ID := 0;
        Active_Target_Weight := 0.0;
        Status_Message := 'Transition Delay';
        
        Transition_Timer(IN := TRUE, PT := T#2S);
        IF Transition_Timer.Q THEN
            Transition_Timer(IN := FALSE);
            Step := (Step - 10) + 1; // Advance to next bin
        END_IF;
        
    16: (* Transition Delay After Last Bin (Bin 6) Closes *)
        Active_Material_ID := 0;
        Active_Bin_ID := 0;
        Active_Target_Weight := 0.0;
        Status_Message := 'Settling Last Bin';
        
        Transition_Timer(IN := TRUE, PT := T#2S);
        IF Transition_Timer.Q THEN
            Transition_Timer(IN := FALSE);
            Step := 7; // Go to post-discharge wait step
        END_IF;

    7: (* Wait 2 Seconds After Closing the Last Bin *)
        Active_Material_ID := 0;
        Active_Bin_ID := 0;
        Active_Target_Weight := 0.0;
        Status_Message := 'Settling Delay';
        Completion_Timer(IN := TRUE, PT := T#2S);
        IF Completion_Timer.Q THEN
            Completion_Timer(IN := FALSE);
            Step := 8; // Proceed to reset last weight
        END_IF;
        
    8: (* Reset bin_last_weight to 0 & Complete *)
        Active_Material_ID := 0;
        Active_Bin_ID := 0;
        Active_Target_Weight := 0.0;
        Status_Message := 'Sequence Completed';
        bin_last_weight := 0.0;
        Sequence_Complete := TRUE;
        
        IF NOT Start_Button THEN
            Step := 0;
            Sequence_Complete := FALSE;
            (* Reset all actual weights at completion once start is released *)
            FOR i := 1 TO 6 DO
                Actual_Weights[i] := 0.0;
            END_FOR;
        END_IF;
END_CASE;

END_FUNCTION_BLOCK

// PLC_AC500_V3/Application/old_version/Semi_Auto_Batching_V12
FUNCTION_BLOCK Semi_Auto_Batching_V12
VAR_INPUT
    Start_Button : BOOL;      // Signal to start/resume the batching sequence
    E_Stop_Active : BOOL;     // Emergency Stop (Pause/Hold signal)
    Reset : BOOL;             // Hard reset sequence back to idle state
    Semi_Auto_Bin_Material_Mapping : ARRAY[1..10] OF INT; // Material index mapping for 10 manual silos
    Semi_Auto_Coarse_To_Fine_speed : ARRAY[1..10] OF REAL; // Cutoff weight thresholds (kg)
    Semi_Auto_Bin_Tolerance : ARRAY[1..10] OF REAL; // Tolerance weight offset values (kg)
END_VAR
VAR_IN_OUT
    load_cell_value : REAL;   // Weight value read/written from load cell
END_VAR
VAR_OUTPUT
    Semi_Auto_Bin : ARRAY[1..10] OF BOOL; // Prompts/indicators for Bins 7..16
    semi_auto_bin_cutoff : ARRAY[1..10] OF BOOL; // Manual pre-cutoff indicators
    semi_auto_bin_motor : ARRAY[1..10] OF BOOL; // Main manual feeder motor outputs
    Actual_Weights : ARRAY[1..10] OF REAL; // Actual weight poured per silo
    Sequence_Complete : BOOL;  // Batch complete flag
    Active_Material_ID : INT;  // Currently active ingredient ID
    Active_Bin_ID : INT;       // Currently active physical Bin ID (7..16)
    Active_Target_Weight : REAL; // Recipe target weight of active bin (with tolerance applied)
    Error_Code : INT;          // Active error code
    Status_Message : STRING;   // Diagnostic text message
END_VAR
VAR
    Step : INT;                // State machine index
    bin_last_weight : REAL;   // Baseline weight snapshot before starting current bin
    actual_bin : REAL;        // Current weight added from active bin
    target_act_bin : REAL;    // Effective target weight to add from the active bin
    cutoff_trigger_weight : REAL; // Calculated target threshold weight
    Paused_By_EStop : BOOL;    // Pause status latch
    
    Mat_Idx : INT;
    i : INT;                  // General loop index
    
    (* TIMERS FOR TRANSITIONS & DELAYS *)
    Transition_Timer : TON;
    Completion_Timer : TON;
    Operator_Timer : TON;
    
    (* SELF-CONTAINED SIMULATION VARIABLES *)
    Simulation_Mode : BOOL;    // Simulation disabled
    Sim_Rate : REAL;
    Sim_Timer : TON;
    Start_Sim_Weight : REAL;
    Discharge_Active : BOOL;
END_VAR

(* Semi-Auto Batching FB V12 with E-Stop Pause & Reset Logic *)

(* 1. HARD RESET INTERLOCK (Resets weights immediately) *)
IF Reset THEN
    FOR i := 1 TO 10 DO
        Semi_Auto_Bin[i] := FALSE;
        semi_auto_bin_cutoff[i] := FALSE;
        semi_auto_bin_motor[i] := FALSE;
        Actual_Weights[i] := 0.0;
    END_FOR;
    Sequence_Complete := FALSE;
    Active_Material_ID := 0;
    Active_Bin_ID := 0;
    Active_Target_Weight := 0.0;
    Error_Code := 0;
    Status_Message := '';
    Paused_By_EStop := FALSE;
    Step := 0;
    
    load_cell_value := 0.0;
    bin_last_weight := 0.0;
    Start_Sim_Weight := 0.0;
    
    Transition_Timer(IN := FALSE);
    Completion_Timer(IN := FALSE);
    Operator_Timer(IN := FALSE);
    Sim_Timer(IN := FALSE);
    RETURN;
END_IF;

(* 2. E-STOP PAUSE / HOLD LOGIC *)
IF E_Stop_Active THEN
    Paused_By_EStop := TRUE;
END_IF;

IF Paused_By_EStop THEN
    (* Suspend all indicators and feeder outputs *)
    FOR i := 1 TO 10 DO
        Semi_Auto_Bin[i] := FALSE;
        semi_auto_bin_cutoff[i] := FALSE;
        semi_auto_bin_motor[i] := FALSE;
    END_FOR;
    
    IF E_Stop_Active THEN
        Status_Message := 'Semi-Auto Paused: Emergency Stop Active!';
    ELSE
        Status_Message := 'Semi-Auto Paused: Press Start to Resume';
        
        (* Resume sequence when Start Button is pressed *)
        IF Start_Button THEN
            Paused_By_EStop := FALSE;
        END_IF;
    END_IF;
    
    (* Freeze simulation and safety timers *)
    Sim_Timer(IN := FALSE);
    Transition_Timer(IN := FALSE);
    Completion_Timer(IN := FALSE);
    Operator_Timer(IN := FALSE);
    RETURN;
END_IF;

(* 3. SELF-CONTAINED SIMULATION WEIGHT MANAGEMENT *)
IF Simulation_Mode THEN
    (* Reset simulation to baseline *)
    IF Step = 0 AND NOT Start_Button AND NOT Sequence_Complete THEN
        load_cell_value := 0.0;
        bin_last_weight := 0.0;
        Start_Sim_Weight := 0.0;
        Sim_Timer(IN := FALSE);
    END_IF;
    
    (* Check if operator is actively pouring *)
    Discharge_Active := FALSE;
    IF Step >= 1 AND Step <= 10 THEN
        Discharge_Active := semi_auto_bin_motor[Step];
    END_IF;
    
    (* Simulate weight gain on the load cell *)
    IF Discharge_Active THEN
        Sim_Timer(IN := TRUE, PT := T#1000S);
        load_cell_value := Start_Sim_Weight + (TIME_TO_REAL(Sim_Timer.ET) / 1000.0) * Sim_Rate;
    ELSE
        Sim_Timer(IN := FALSE);
        Start_Sim_Weight := load_cell_value;
    END_IF;
END_IF;


(* 4. RECIPE SEQUENCE START *)
IF Step = 0 AND Start_Button THEN
    Step := 1;
    bin_last_weight := load_cell_value;
    Sequence_Complete := FALSE;
    Error_Code := 0;
    Status_Message := 'Semi-Auto Pour Started';
    Active_Target_Weight := 0.0;
    (* Clear actual weights on start *)
    FOR i := 1 TO 10 DO
        Actual_Weights[i] := 0.0;
        Semi_Auto_Bin[i] := FALSE;
        semi_auto_bin_cutoff[i] := FALSE;
        semi_auto_bin_motor[i] := FALSE;
    END_FOR;
END_IF;


(* 5. SEQUENCE CONTROL STATE MACHINE *)
CASE Step OF
    0:
        Active_Material_ID := 0;
        Active_Bin_ID := 0;
        Active_Target_Weight := 0.0;
        IF Error_Code = 0 THEN Status_Message := 'Semi-Auto Idle'; END_IF;
        
    1..10: (* Prompts Silos 7 to 16 *)
        Mat_Idx := Semi_Auto_Bin_Material_Mapping[Step];
        
        (* Skip this step instantly if material mapping is 0 OR target weight is 0.0 kg *)
        IF Mat_Idx = 0 OR (Mat_Idx <= 20 AND GVL.Recipe_Weights[Mat_Idx] = 0.0) THEN
            Step := Step + 1;
        ELSE
            (* Calculate effective target weight (Looked up Target - Tolerance) *)
            target_act_bin := GVL.Recipe_Weights[Mat_Idx] - Semi_Auto_Bin_Tolerance[Step];
            Active_Target_Weight := target_act_bin;
            
            (* Calculate weight added by current active bin *)
            actual_bin := load_cell_value - bin_last_weight;
            Actual_Weights[Step] := actual_bin;
            
            (* Calculate cutoff trigger threshold *)
            cutoff_trigger_weight := target_act_bin - Semi_Auto_Coarse_To_Fine_speed[Step];
            
            Active_Material_ID := Mat_Idx;
            Active_Bin_ID := Step;
            Status_Message := 'Semi-Auto Pouring Active';
            
            (* COARSE/FINE FEED TRANSITIONS WITH TOLERANCE OFFSETS *)
            IF actual_bin < cutoff_trigger_weight THEN
                (* Phase 1: Coarse Feed *)
                Semi_Auto_Bin[Step] := TRUE;
                semi_auto_bin_cutoff[Step] := FALSE;
                semi_auto_bin_motor[Step] := TRUE;
            ELSIF actual_bin < target_act_bin THEN
                (* Phase 2: Fine Feed *)
                Semi_Auto_Bin[Step] := FALSE;
                semi_auto_bin_cutoff[Step] := TRUE;
                semi_auto_bin_motor[Step] := TRUE;
            ELSE
                (* Phase 3: Completed (All OFF) *)
                Semi_Auto_Bin[Step] := FALSE;
                semi_auto_bin_cutoff[Step] := FALSE;
                semi_auto_bin_motor[Step] := FALSE;
                bin_last_weight := load_cell_value;
                Active_Target_Weight := 0.0;
                Step := 10 + Step; // Offset to separate transition states
            END_IF;
            
            (* RUNTIME CHECKS *)
            (* Check 21 & 22: Scale Limits *)
            IF load_cell_value > 500.0 THEN
                Error_Code := 21;
                Status_Message := 'Error 21: Scale Overloaded!';
                Sequence_Complete := TRUE; // Mark complete on halt
                Paused_By_EStop := TRUE;
            ELSIF load_cell_value < 0.0 THEN
                Error_Code := 22;
                Status_Message := 'Error 22: Scale Underloaded/Fault!';
                Sequence_Complete := TRUE; // Mark complete on halt
                Paused_By_EStop := TRUE;
            END_IF;
            
            (* Check 30: Operator Timeout *)
            Operator_Timer(IN := semi_auto_bin_motor[Step], PT := T#300S);
            IF Operator_Timer.Q THEN
                Error_Code := 30;
                Status_Message := 'Error 30: Semi-Auto Operator Timeout!';
                Sequence_Complete := TRUE; // Mark complete on halt
                Paused_By_EStop := TRUE;
            END_IF;
        END_IF;

    11..19: (* Transition Delays (Between Bins) *)
        Active_Material_ID := 0;
        Active_Bin_ID := 0;
        Active_Target_Weight := 0.0;
        Status_Message := 'Transition Delay';
        Transition_Timer(IN := TRUE, PT := T#2S);
        IF Transition_Timer.Q THEN
            Transition_Timer(IN := FALSE);
            Step := (Step - 10) + 1; // Advance to next bin
        END_IF;
        
    20: (* Transition Delay After Last Bin (Bin 10) Closes *)
        Active_Material_ID := 0;
        Active_Bin_ID := 0;
        Active_Target_Weight := 0.0;
        Status_Message := 'Settling Last Bin';
        Transition_Timer(IN := TRUE, PT := T#2S);
        IF Transition_Timer.Q THEN
            Transition_Timer(IN := FALSE);
            Step := 30; // Go to post-discharge wait step (State 30)
        END_IF;

    30: (* Wait 2 Seconds After Closing the Last Bin *)
        Active_Material_ID := 0;
        Active_Bin_ID := 0;
        Active_Target_Weight := 0.0;
        Status_Message := 'Settling Delay';
        Completion_Timer(IN := TRUE, PT := T#2S);
        IF Completion_Timer.Q THEN
            Completion_Timer(IN := FALSE);
            Step := 40; // Proceed to reset last weight (State 40)
        END_IF;
        
    40: (* Reset bin_last_weight to 0 & Complete *)
        Active_Material_ID := 0;
        Active_Bin_ID := 0;
        Active_Target_Weight := 0.0;
        Status_Message := 'Sequence Completed';
        bin_last_weight := 0.0;
        Sequence_Complete := TRUE;
        
        IF NOT Start_Button THEN
            Step := 0;
            Sequence_Complete := FALSE;
            (* Reset all actual weights at completion once start is released *)
            FOR i := 1 TO 10 DO
                Actual_Weights[i] := 0.0;
            END_FOR;
        END_IF;
END_CASE;

END_FUNCTION_BLOCK

// PLC_AC500_V3/Application/old_version/batching12
PROGRAM batching12
VAR
    Auto_Ctrl : Auto_Batching_V12;
    Semi_Auto_Ctrl : Semi_Auto_Batching_V12;
    
    (* Sub-Block Diagnostic Indicators (not in GVL) *)
    Auto_Active_Target : REAL; // Active Target Weight for Auto (displays GVL setpoint - Tolerance)
    Auto_Err : INT;
    Auto_Msg : STRING;
    
    Semi_Auto_Active_Target : REAL; // Active Target Weight for Semi-Auto (displays GVL setpoint - Tolerance)
    Semi_Auto_Err : INT;
    Semi_Auto_Msg : STRING;
    
    (* Process Outputs *)
    Auto_Bin : ARRAY[1..6] OF BOOL; // Valve control outputs (Coarse)
    auto_bin_cutoff : ARRAY[1..6] OF BOOL; // Cutoff indicators (Fine)
    auto_bin_motor : ARRAY[1..6] OF BOOL; // Conveyor/feeder motor outputs
    
    Semi_Auto_Bin : ARRAY[1..10] OF BOOL; // Prompt indicators (Coarse)
    semi_auto_bin_cutoff : ARRAY[1..10] OF BOOL; // Cutoff indicators (Fine)
    semi_auto_bin_motor : ARRAY[1..10] OF BOOL; // Conveyor/feeder motor outputs
    
    Auto_Weights : ARRAY[1..6] OF REAL;
    Semi_Auto_Weights : ARRAY[1..10] OF REAL;
    
    Auto_Complete : BOOL;
    Semi_Auto_Complete : BOOL;
    
    (* Repetitive Cycle Status (not in GVL) *)
    Completed_Batch_Cycles : INT;      // Total completed batch cycle loops
    All_Cycles_Complete : BOOL;         // Indicator for full set completion
    
    (* Diagnostics & Interlocks (not in GVL) *)
    Status_Message : STRING;
    
    i : INT;
    j : INT;
    Duplicate_Found : BOOL;
    Invalid_Material_Range : BOOL;
    Weight_Limit_Error : BOOL;
    
    (* Cycle Manager state variables *)
    Cycle_Manager_State : INT;         // State index for loop management
    Internal_FB_Start : BOOL;          // Controlled command to restart sub-blocks
END_VAR

(* 1. STARTUP CONFIGURATION AND WEIGHT CHECKS *)
Duplicate_Found := FALSE;
Invalid_Material_Range := FALSE;
Weight_Limit_Error := FALSE;

FOR i := 1 TO 6 DO
    (* Check 2: Out of Range (Auto) *)
    IF GVL.Auto_Bin_Material_Mapping[i] < 0 OR GVL.Auto_Bin_Material_Mapping[i] > 20 THEN
        Invalid_Material_Range := TRUE;
    END_IF;
    
    (* Check 1: Duplicate Cross-Array Material ID *)
    IF GVL.Auto_Bin_Material_Mapping[i] <> 0 AND GVL.Auto_Bin_Material_Mapping[i] <= 20 THEN
        FOR j := 1 TO 10 DO
            IF GVL.Auto_Bin_Material_Mapping[i] = GVL.Semi_Auto_Bin_Material_Mapping[j] THEN
                Duplicate_Found := TRUE;
            END_IF;
        END_FOR;
    END_IF;
    
    (* Check 3: Recipe weight is less than Cutoff + Tolerance *)
    IF GVL.Auto_Bin_Material_Mapping[i] <> 0 AND GVL.Auto_Bin_Material_Mapping[i] <= 20 THEN
        IF GVL.Recipe_Weights[GVL.Auto_Bin_Material_Mapping[i]] > 0.0 THEN
            IF GVL.Recipe_Weights[GVL.Auto_Bin_Material_Mapping[i]] < (GVL.Auto_Coarse_To_Fine_speed[i] + GVL.Auto_Bin_Tolerance[i]) THEN
                Weight_Limit_Error := TRUE;
            END_IF;
        END_IF;
    END_IF;
END_FOR;

FOR j := 1 TO 10 DO
    (* Check 2: Out of Range (Semi-Auto) *)
    IF GVL.Semi_Auto_Bin_Material_Mapping[j] < 0 OR GVL.Semi_Auto_Bin_Material_Mapping[j] > 20 THEN
        Invalid_Material_Range := TRUE;
    END_IF;
    
    (* Check 3: Recipe weight check (Semi-Auto) *)
    IF GVL.Semi_Auto_Bin_Material_Mapping[j] <> 0 AND GVL.Semi_Auto_Bin_Material_Mapping[j] <= 20 THEN
        IF GVL.Recipe_Weights[GVL.Semi_Auto_Bin_Material_Mapping[j]] > 0.0 THEN
            IF GVL.Recipe_Weights[GVL.Semi_Auto_Bin_Material_Mapping[j]] < (GVL.Semi_Auto_Coarse_To_Fine_speed[j] + GVL.Semi_Auto_Bin_Tolerance[j]) THEN
                Weight_Limit_Error := TRUE;
            END_IF;
        END_IF;
    END_IF;
END_FOR;

(* Configuration Error Resolution *)
IF Duplicate_Found THEN
    GVL.Error_Code := 1;
    Status_Message := 'Error 1: Duplicate Material ID mapped in Auto and Semi-Auto!';
ELSIF Invalid_Material_Range THEN
    GVL.Error_Code := 2;
    Status_Message := 'Error 2: Material Index configuration out of range (1..20)!';
ELSIF Weight_Limit_Error THEN
    GVL.Error_Code := 3;
    Status_Message := 'Error 3: Recipe weight is less than Cutoff + Tolerance!';
ELSE
    IF GVL.Error_Code <= 3 THEN
        GVL.Error_Code := 0;
    END_IF;
END_IF;

(* Abort/Clear arrays if Configuration error is active or Hard Reset is pressed *)
IF (GVL.Error_Code >= 1 AND GVL.Error_Code <= 3) OR GVL.Reset THEN
    FOR i := 1 TO 6 DO 
        Auto_Bin[i] := FALSE; 
        auto_bin_cutoff[i] := FALSE; 
        auto_bin_motor[i] := FALSE; 
        Auto_Weights[i] := 0.0;
    END_FOR;
    
    FOR i := 1 TO 10 DO 
        Semi_Auto_Bin[i] := FALSE; 
        semi_auto_bin_cutoff[i] := FALSE; 
        semi_auto_bin_motor[i] := FALSE; 
        Semi_Auto_Weights[i] := 0.0;
    END_FOR;
    
    Internal_FB_Start := FALSE;
    Auto_Ctrl(Start_Button := FALSE, E_Stop_Active := FALSE, Reset := GVL.Reset, load_cell_value := GVL.load_cell_auto);
    Semi_Auto_Ctrl(Start_Button := FALSE, E_Stop_Active := FALSE, Reset := GVL.Reset, load_cell_value := GVL.load_cell_semi_auto);
    
    Auto_Active_Target := 0.0;
    Semi_Auto_Active_Target := 0.0;
    
    Auto_Complete := TRUE;
    Semi_Auto_Complete := TRUE;
    All_Cycles_Complete := TRUE;
    
    GVL.Cycle_Hold_Active := FALSE;
    GVL.Run := FALSE;
    Cycle_Manager_State := 0;
    
    IF GVL.Reset THEN
        GVL.Error_Code := 0;
        GVL.Current_Batch_Cycle := 0;
        Completed_Batch_Cycles := 0;
        Status_Message := 'System Reset Activated';
        Auto_Complete := FALSE;
        Semi_Auto_Complete := FALSE;
        All_Cycles_Complete := FALSE;
        
        GVL.Auto_Active_Mat := 0;
        GVL.Auto_Active_Bin := 0;
        GVL.Semi_Auto_Active_Mat := 0;
        GVL.Semi_Auto_Active_Bin := 0;
    END_IF;
    RETURN;
END_IF;


(* 2. REPETITIVE CYCLE MANAGER STATE MACHINE WITH HOLD RELEASE *)
CASE Cycle_Manager_State OF
    0: (* IDLE STATE *)
        Internal_FB_Start := FALSE;
        All_Cycles_Complete := FALSE;
        GVL.Cycle_Hold_Active := FALSE;
        GVL.Run := FALSE;
        IF GVL.Error_Code = 0 THEN Status_Message := 'System Ready'; END_IF;
        
        IF GVL.Start_Button THEN
            GVL.Current_Batch_Cycle := 1;
            Completed_Batch_Cycles := 0;
            
            (* Explicitly reset latch flags so FBs can run fresh *)
            Auto_Complete := FALSE;
            Semi_Auto_Complete := FALSE;
            
            GVL.Run := TRUE;
            Cycle_Manager_State := 1;
        END_IF;
        
    1: (* RUN STATE (Run Sub-Blocks) *)
        Internal_FB_Start := TRUE;
        GVL.Run := TRUE;
        Status_Message := CONCAT('Running Batch Cycle ', INT_TO_STRING(GVL.Current_Batch_Cycle));
        
        (* Monitor completion of active step *)
        IF Auto_Complete AND Semi_Auto_Complete THEN
            Cycle_Manager_State := 2;
        END_IF;
        
    2: (* CHECK REPEAT CYCLE STATE *)
        Completed_Batch_Cycles := GVL.Current_Batch_Cycle;
        GVL.Run := TRUE;
        
        (* Block cycle repeat in case of active error *)
        IF GVL.Current_Batch_Cycle < GVL.Target_Batch_Cycles AND GVL.Error_Code = 0 THEN
            (* Hold cycle loop progression *)
            GVL.Cycle_Hold_Active := TRUE;
            Cycle_Manager_State := 5; // Go to hold wait state
        else
            (* All loop cycles complete *)
            Cycle_Manager_State := 4;
        END_IF;
        
    5: (* PAUSED BETWEEN CYCLES *)
        Internal_FB_Start := TRUE; // Keep FBs active in finished step state
        GVL.Run := TRUE;
        Status_Message := CONCAT('Cycle ', CONCAT(INT_TO_STRING(GVL.Current_Batch_Cycle), ' Complete. Waiting to Release.'));
        
        (* Operator toggles hold status back to FALSE to proceed *)
        IF NOT GVL.Cycle_Hold_Active THEN
            Cycle_Manager_State := 3; // Go to auto-reset pulse
        END_IF;
        
    3: (* AUTO-RESET PULSE (Pulse Start command low to reset state machines) *)
        Internal_FB_Start := FALSE;
        GVL.Run := TRUE;
        Status_Message := 'Resetting Sequence for Next Cycle';
        
        (* Verify sub-blocks have fully reset to idle step *)
        IF NOT Auto_Complete AND NOT Semi_Auto_Complete THEN
            GVL.Current_Batch_Cycle := GVL.Current_Batch_Cycle + 1;
            Cycle_Manager_State := 1; // Start next cycle
        END_IF;
        
    4: (* SEQUENCE FULLY COMPLETED STATE *)
        Internal_FB_Start := FALSE;
        All_Cycles_Complete := TRUE;
        GVL.Run := FALSE;
        Status_Message := 'All Batch Cycles Completed';
        
        IF NOT GVL.Start_Button THEN
            Cycle_Manager_State := 0;
        END_IF;
END_CASE;


(* 3. CONCURRENT EXECUTION OF FB INSTANCES *)
Auto_Ctrl(
    Start_Button := Internal_FB_Start,
    E_Stop_Active := GVL.E_Stop_Active,
    Reset := GVL.Reset,
    load_cell_value := GVL.load_cell_auto,
    Auto_Bin_Material_Mapping := GVL.Auto_Bin_Material_Mapping,
    Auto_Coarse_To_Fine_speed := GVL.Auto_Coarse_To_Fine_speed,
    Auto_Bin_Tolerance := GVL.Auto_Bin_Tolerance,
    Auto_Bin => Auto_Bin,
    auto_bin_cutoff => auto_bin_cutoff,
    auto_bin_motor => auto_bin_motor,
    Actual_Weights => Auto_Weights,
    Sequence_Complete => Auto_Complete,
    Active_Material_ID => GVL.Auto_Active_Mat,
    Active_Bin_ID => GVL.Auto_Active_Bin,
    Active_Target_Weight => Auto_Active_Target,
    Error_Code => Auto_Err,
    Status_Message => Auto_Msg
);

Semi_Auto_Ctrl(
    Start_Button := Internal_FB_Start,
    E_Stop_Active := GVL.E_Stop_Active,
    Reset := GVL.Reset,
    load_cell_value := GVL.load_cell_semi_auto,
    Semi_Auto_Bin_Material_Mapping := GVL.Semi_Auto_Bin_Material_Mapping,
    Semi_Auto_Coarse_To_Fine_speed := GVL.Semi_Auto_Coarse_To_Fine_speed,
    Semi_Auto_Bin_Tolerance := GVL.Semi_Auto_Bin_Tolerance,
    Semi_Auto_Bin => Semi_Auto_Bin,
    semi_auto_bin_cutoff => semi_auto_bin_cutoff,
    semi_auto_bin_motor => semi_auto_bin_motor,
    Actual_Weights => Semi_Auto_Weights,
    Sequence_Complete => Semi_Auto_Complete,
    Active_Material_ID => GVL.Semi_Auto_Active_Mat,
    Active_Bin_ID => GVL.Semi_Auto_Active_Bin,
    Active_Target_Weight => Semi_Auto_Active_Target,
    Error_Code => Semi_Auto_Err,
    Status_Message => Semi_Auto_Msg
);

(* Runtime Error Mapping & Aggregation *)
IF Auto_Err <> 0 THEN
    GVL.Error_Code := Auto_Err;
    Status_Message := CONCAT('Auto Error: ', Auto_Msg);
    (* Wherever it stops, completion outputs must register TRUE *)
    Auto_Complete := TRUE;
    Semi_Auto_Complete := TRUE;
    All_Cycles_Complete := TRUE;
    GVL.Run := FALSE;
ELSIF Semi_Auto_Err <> 0 THEN
    GVL.Error_Code := Semi_Auto_Err;
    Status_Message := CONCAT('Semi-Auto Error: ', Semi_Auto_Msg);
    (* Wherever it stops, completion outputs must register TRUE *)
    Auto_Complete := TRUE;
    Semi_Auto_Complete := TRUE;
    All_Cycles_Complete := TRUE;
    GVL.Run := FALSE;
ELSIF Cycle_Manager_State = 0 THEN
    GVL.Error_Code := 0;
END_IF;

END_PROGRAM

// PLC_AC500_V3/Application/old_version/Auto_Batching_V13
FUNCTION_BLOCK Auto_Batching_V13
VAR_INPUT
    Start_Button : BOOL;      // Signal to start/resume the batching sequence
    E_Stop_Active : BOOL;     // Emergency Stop (Pause/Hold signal)
    Reset : BOOL;             // Hard reset sequence trigger
    Auto_Bin_Material_Mapping : ARRAY[1..6] OF INT; // Material index mapping for 6 bins
    Auto_Coarse_To_Fine_speed : ARRAY[1..6] OF REAL; // Cutoff weight thresholds (kg)
    Auto_Bin_Tolerance : ARRAY[1..6] OF REAL; // Tolerance weight offset values (kg)
    Inter_Bin_Delay : TIME;   // Global inter-bin delay time
    Excess_Allowed : BOOL;    // Global toggle: TRUE = skip excess check, FALSE = trigger alarm & hold
END_VAR
VAR_IN_OUT
    load_cell_value : REAL;   // Weight value read/written from load cell
END_VAR
VAR_OUTPUT
    Auto_Bin : ARRAY[1..6] OF BOOL; // Coarse feed valve outputs
    auto_bin_cutoff : ARRAY[1..6] OF BOOL; // Fine feed cutoff trigger indicators
    auto_bin_motor : ARRAY[1..6] OF BOOL; // Main conveyor motor outputs
    Actual_Weights : ARRAY[1..6] OF REAL; // Actual weight poured per silo
    Sequence_Complete : BOOL;  // Batch complete flag
    Active_Material_ID : INT;  // Currently active ingredient ID
    Active_Bin_ID : INT;       // Currently active physical Bin ID (1..6)
    Active_Target_Weight : REAL; // Recipe target weight of active bin
    Active_Live_Weight : REAL; // Live tared weight poured from active bin
    Excess_Alarm : BOOL;       // Excess weight alarm output
    Error_Code : INT;          // Active error code
    Status_Message : STRING;   // Diagnostic text message
END_VAR
VAR
    Step : INT;                // State machine index (0: Idle, 1..6: Pour, 7: Settling, 8: Complete)
    bin_last_weight : REAL;   // Baseline weight snapshot before starting current bin
    actual_bin : REAL;        // Current weight added from active bin
    target_weight : REAL;     // Target recipe weight
    cutoff_trigger_weight : REAL; // Calculated cutoff trigger threshold (Target - Cutoff)
    min_tol_weight : REAL;    // Minimum allowable tolerance (Target - Tol)
    max_tol_weight : REAL;    // Maximum allowable tolerance (Target + Tol)
    Paused_By_EStop : BOOL;    // Pause status latch
    Effective_Delay : TIME;   // Resolved delay time (defaults to T#2S if T#0S configured)
    
    Mat_Idx : INT;
    i : INT;                  // General loop index
    
    (* TIMERS FOR TRANSITIONS & DELAYS *)
    Transition_Timer : TON;
    Completion_Timer : TON;
    
    (* SELF-CONTAINED SIMULATION VARIABLES *)
    Simulation_Mode : BOOL;    // Simulation disabled for physical PLC use
    Sim_Rate : REAL;
    Sim_Timer : TON;
    Start_Sim_Weight : REAL;
    Discharge_Active : BOOL;
END_VAR

(* Auto Batching FB V13 with Real-Time Instant Excess Verification & Clean Multi-Cycle Reset *)

Effective_Delay := Inter_Bin_Delay;
IF Effective_Delay = T#0S THEN
    Effective_Delay := T#2S;
END_IF;

(* 1. HARD RESET INTERLOCK *)
IF Reset THEN
    FOR i := 1 TO 6 DO
        Auto_Bin[i] := FALSE;
        auto_bin_cutoff[i] := FALSE;
        auto_bin_motor[i] := FALSE;
        Actual_Weights[i] := 0.0;
    END_FOR;
    Sequence_Complete := FALSE;
    Active_Material_ID := 0;
    Active_Bin_ID := 0;
    Active_Target_Weight := 0.0;
    Active_Live_Weight := 0.0;
    Excess_Alarm := FALSE;
    Error_Code := 0;
    Status_Message := '';
    Paused_By_EStop := FALSE;
    Step := 0;
    
    bin_last_weight := 0.0;
    Start_Sim_Weight := 0.0;
    
    Transition_Timer(IN := FALSE);
    Completion_Timer(IN := FALSE);
    Sim_Timer(IN := FALSE);
    RETURN;
END_IF;

(* 2. E-STOP PAUSE / HOLD LOGIC *)
IF E_Stop_Active THEN
    Paused_By_EStop := TRUE;
END_IF;

IF Paused_By_EStop THEN
    FOR i := 1 TO 6 DO
        Auto_Bin[i] := FALSE;
        auto_bin_cutoff[i] := FALSE;
        auto_bin_motor[i] := FALSE;
    END_FOR;
    
    IF E_Stop_Active THEN
        Status_Message := 'Auto Paused: Emergency Stop Active!';
    ELSE
        Status_Message := 'Auto Paused: Press Start to Resume';
        IF Start_Button THEN
            Paused_By_EStop := FALSE;
        END_IF;
    END_IF;
    
    Sim_Timer(IN := FALSE);
    Transition_Timer(IN := FALSE);
    Completion_Timer(IN := FALSE);
    RETURN;
END_IF;

(* 3. SIMULATION WEIGHT MANAGEMENT (WHEN ENABLED) *)
IF Simulation_Mode THEN
    IF Step = 0 AND NOT Start_Button AND NOT Sequence_Complete THEN
        load_cell_value := 0.0;
        bin_last_weight := 0.0;
        Start_Sim_Weight := 0.0;
        Sim_Timer(IN := FALSE);
    END_IF;
    
    Discharge_Active := FALSE;
    IF Step >= 1 AND Step <= 6 THEN
        Discharge_Active := auto_bin_motor[Step];
    END_IF;
    
    IF Discharge_Active THEN
        Sim_Timer(IN := TRUE, PT := T#1000S);
        load_cell_value := Start_Sim_Weight + (TIME_TO_REAL(Sim_Timer.ET) / 1000.0) * Sim_Rate;
    ELSE
        Sim_Timer(IN := FALSE);
        Start_Sim_Weight := load_cell_value;
    END_IF;
END_IF;

(* 4. RECIPE SEQUENCE START & CYCLIC RESET *)
IF Step = 0 AND Start_Button THEN
    Step := 1;
    bin_last_weight := load_cell_value; (* Snapshot relative tare at whatever weight scale is *)
    Sequence_Complete := FALSE;
    Excess_Alarm := FALSE;
    Error_Code := 0;
    Status_Message := 'Auto Pour Started';
    Active_Target_Weight := 0.0;
    Active_Live_Weight := 0.0;
    FOR i := 1 TO 6 DO
        Actual_Weights[i] := 0.0;
        Auto_Bin[i] := FALSE;
        auto_bin_cutoff[i] := FALSE;
        auto_bin_motor[i] := FALSE;
    END_FOR;
END_IF;

(* 5. SEQUENCE CONTROL STATE MACHINE *)
CASE Step OF
    0:
        Active_Material_ID := 0;
        Active_Bin_ID := 0;
        Active_Target_Weight := 0.0;
        Active_Live_Weight := 0.0;
        Excess_Alarm := FALSE;
        Sequence_Complete := FALSE;
        FOR i := 1 TO 6 DO
            Auto_Bin[i] := FALSE;
            auto_bin_cutoff[i] := FALSE;
            auto_bin_motor[i] := FALSE;
        END_FOR;
        IF Error_Code = 0 THEN Status_Message := 'Auto Idle'; END_IF;
        
    1..6: (* DISCHARGE SILOS 1 TO 6 *)
        Mat_Idx := Auto_Bin_Material_Mapping[Step];
        
        (* Skip this step instantly if material mapping is 0 OR target weight is 0.0 kg *)
        IF Mat_Idx = 0 OR (Mat_Idx <= 20 AND GVL.Recipe_Weights[Mat_Idx] = 0.0) THEN
            IF Step = 6 THEN
                Step := 7; (* Transition directly to final settling delay *)
            ELSE
                Step := Step + 1;
            END_IF;
        ELSE
            target_weight := GVL.Recipe_Weights[Mat_Idx];
            cutoff_trigger_weight := target_weight - Auto_Coarse_To_Fine_speed[Step];
            min_tol_weight := target_weight - Auto_Bin_Tolerance[Step];
            max_tol_weight := target_weight + Auto_Bin_Tolerance[Step];
            
            Active_Target_Weight := target_weight;
            actual_bin := load_cell_value - bin_last_weight;
            Actual_Weights[Step] := actual_bin;
            Active_Live_Weight := actual_bin; (* Live tared weight of active bin *)
            
            Active_Material_ID := Mat_Idx;
            Active_Bin_ID := Step;
            
            (* Scale Overload Protection *)
            IF load_cell_value > 500.0 THEN
                Error_Code := 21;
                Status_Message := 'Error 21: Scale Overloaded!';
                Sequence_Complete := TRUE;
                Paused_By_EStop := TRUE;
            END_IF;
            
            (* Real-Time Feed & Instant Excess Alarm *)
            IF actual_bin < cutoff_trigger_weight THEN
                (* Coarse Feed *)
                Auto_Bin[Step] := TRUE;
                auto_bin_cutoff[Step] := FALSE;
                auto_bin_motor[Step] := TRUE;
                Excess_Alarm := FALSE;
                Status_Message := 'Auto Pouring (Coarse Feed)';
                
            ELSIF actual_bin < min_tol_weight THEN
                (* Fine Feed *)
                Auto_Bin[Step] := FALSE;
                auto_bin_cutoff[Step] := TRUE;
                auto_bin_motor[Step] := TRUE;
                Excess_Alarm := FALSE;
                Status_Message := 'Auto Pouring (Fine Feed)';
                
            ELSIF actual_bin > max_tol_weight THEN
                (* Excess Weight -> Instant Alarm, No Delay! *)
                Auto_Bin[Step] := FALSE;
                auto_bin_cutoff[Step] := FALSE;
                auto_bin_motor[Step] := FALSE;
                
                IF Excess_Allowed THEN
                    Excess_Alarm := FALSE;
                    Status_Message := 'Excess Weight Allowed: Advancing';
                    bin_last_weight := load_cell_value;
                    Active_Target_Weight := 0.0;
                    Active_Live_Weight := 0.0;
                    IF Step = 6 THEN
                        Step := 7;
                    ELSE
                        Step := Step + 1;
                    END_IF;
                ELSE
                    Excess_Alarm := TRUE; (* Immediate Trigger! *)
                    Status_Message := 'Excess Alarm: Weight above max tolerance! Reduce weight.';
                END_IF;
                
            ELSE
                (* In Tolerance Window [Min_Tol .. Max_Tol] *)
                Auto_Bin[Step] := FALSE;
                auto_bin_cutoff[Step] := FALSE;
                auto_bin_motor[Step] := FALSE;
                Excess_Alarm := FALSE;
                bin_last_weight := load_cell_value;
                Active_Target_Weight := 0.0;
                Active_Live_Weight := 0.0;
                
                IF Step = 6 THEN
                    Step := 7;
                ELSE
                    Step := Step + 1;
                END_IF;
            END_IF;
        END_IF;

    7: (* POST-SEQUENCE FINAL SETTLING DELAY *)
        Active_Material_ID := 0;
        Active_Bin_ID := 0;
        Active_Target_Weight := 0.0;
        Active_Live_Weight := 0.0;
        Excess_Alarm := FALSE;
        Status_Message := 'Final Settling Delay';
        Completion_Timer(IN := TRUE, PT := Effective_Delay);
        IF Completion_Timer.Q THEN
            Completion_Timer(IN := FALSE);
            Step := 8;
        END_IF;
        
    8: (* COMPLETE *)
        Active_Material_ID := 0;
        Active_Bin_ID := 0;
        Active_Target_Weight := 0.0;
        Active_Live_Weight := 0.0;
        Excess_Alarm := FALSE;
        Status_Message := 'Sequence Completed';
        Sequence_Complete := TRUE;
        
        IF NOT Start_Button THEN
            Step := 0;
            Sequence_Complete := FALSE;
            FOR i := 1 TO 6 DO
                Actual_Weights[i] := 0.0;
            END_FOR;
        END_IF;
END_CASE;

END_FUNCTION_BLOCK

// PLC_AC500_V3/Application/old_version/Semi_Auto_Batching_V13
FUNCTION_BLOCK Semi_Auto_Batching_V13
VAR_INPUT
    Start_Button : BOOL;      // Signal to start/resume the batching sequence
    E_Stop_Active : BOOL;     // Emergency Stop (Pause/Hold signal)
    Reset : BOOL;             // Hard reset sequence trigger
    Semi_Auto_Bin_Material_Mapping : ARRAY[1..10] OF INT; // Material index mapping for 10 manual silos
    Semi_Auto_Coarse_To_Fine_speed : ARRAY[1..10] OF REAL; // Cutoff weight thresholds (kg)
    Semi_Auto_Bin_Tolerance : ARRAY[1..10] OF REAL; // Tolerance weight offset values (kg)
    Inter_Bin_Delay : TIME;   // Global inter-bin delay time
    Excess_Allowed : BOOL;    // Global toggle: TRUE = skip excess check, FALSE = trigger alarm & hold
END_VAR
VAR_IN_OUT
    load_cell_value : REAL;   // Weight value read/written from load cell
END_VAR
VAR_OUTPUT
    Semi_Auto_Bin : ARRAY[1..10] OF BOOL; // Prompts/indicators for Bins 1..10
    semi_auto_bin_cutoff : ARRAY[1..10] OF BOOL; // Manual pre-cutoff indicators
    semi_auto_bin_motor : ARRAY[1..10] OF BOOL; // Main manual feeder motor outputs
    Actual_Weights : ARRAY[1..10] OF REAL; // Actual weight poured per silo
    Sequence_Complete : BOOL;  // Batch complete flag
    Active_Material_ID : INT;  // Currently active ingredient ID
    Active_Bin_ID : INT;       // Currently active physical Bin ID (1..10)
    Active_Target_Weight : REAL; // Recipe target weight of active bin
    Active_Live_Weight : REAL; // Live tared weight poured from active bin
    Excess_Alarm : BOOL;       // Excess weight alarm output
    Error_Code : INT;          // Active error code
    Status_Message : STRING;   // Diagnostic text message
END_VAR
VAR
    Step : INT;                // State machine index (0: Idle, 1..10: Pour, 31: Settling, 32: Complete)
    bin_last_weight : REAL;   // Baseline weight snapshot before starting current bin
    actual_bin : REAL;        // Current weight added from active bin
    target_weight : REAL;     // Target recipe weight
    cutoff_trigger_weight : REAL; // Calculated target threshold weight (Target - Cutoff)
    min_tol_weight : REAL;    // Minimum allowable tolerance (Target - Tol)
    max_tol_weight : REAL;    // Maximum allowable tolerance (Target + Tol)
    Paused_By_EStop : BOOL;    // Pause status latch
    Effective_Delay : TIME;   // Resolved delay time (defaults to T#2S if T#0S configured)
    
    Mat_Idx : INT;
    i : INT;                  // General loop index
    
    (* TIMERS FOR TRANSITIONS & DELAYS *)
    Transition_Timer : TON;
    Completion_Timer : TON;
    
    (* SELF-CONTAINED SIMULATION VARIABLES *)
    Simulation_Mode : BOOL;    // Simulation disabled for physical PLC use
    Sim_Rate : REAL;
    Sim_Timer : TON;
    Start_Sim_Weight : REAL;
    Discharge_Active : BOOL;
END_VAR

(* Semi-Auto Batching FB V13 with Real-Time Instant Excess Verification & Clean Multi-Cycle Reset *)

Effective_Delay := Inter_Bin_Delay;
IF Effective_Delay = T#0S THEN
    Effective_Delay := T#2S;
END_IF;

(* 1. HARD RESET INTERLOCK *)
IF Reset THEN
    FOR i := 1 TO 10 DO
        Semi_Auto_Bin[i] := FALSE;
        semi_auto_bin_cutoff[i] := FALSE;
        semi_auto_bin_motor[i] := FALSE;
        Actual_Weights[i] := 0.0;
    END_FOR;
    Sequence_Complete := FALSE;
    Active_Material_ID := 0;
    Active_Bin_ID := 0;
    Active_Target_Weight := 0.0;
    Active_Live_Weight := 0.0;
    Excess_Alarm := FALSE;
    Error_Code := 0;
    Status_Message := '';
    Paused_By_EStop := FALSE;
    Step := 0;
    
    bin_last_weight := 0.0;
    Start_Sim_Weight := 0.0;
    
    Transition_Timer(IN := FALSE);
    Completion_Timer(IN := FALSE);
    Sim_Timer(IN := FALSE);
    RETURN;
END_IF;

(* 2. E-STOP PAUSE / HOLD LOGIC *)
IF E_Stop_Active THEN
    Paused_By_EStop := TRUE;
END_IF;

IF Paused_By_EStop THEN
    FOR i := 1 TO 10 DO
        Semi_Auto_Bin[i] := FALSE;
        semi_auto_bin_cutoff[i] := FALSE;
        semi_auto_bin_motor[i] := FALSE;
    END_FOR;
    
    IF E_Stop_Active THEN
        Status_Message := 'Semi-Auto Paused: Emergency Stop Active!';
    ELSE
        Status_Message := 'Semi-Auto Paused: Press Start to Resume';
        IF Start_Button THEN
            Paused_By_EStop := FALSE;
        END_IF;
    END_IF;
    
    Sim_Timer(IN := FALSE);
    Transition_Timer(IN := FALSE);
    Completion_Timer(IN := FALSE);
    RETURN;
END_IF;

(* 3. SIMULATION WEIGHT MANAGEMENT (WHEN ENABLED) *)
IF Simulation_Mode THEN
    IF Step = 0 AND NOT Start_Button AND NOT Sequence_Complete THEN
        load_cell_value := 0.0;
        bin_last_weight := 0.0;
        Start_Sim_Weight := 0.0;
        Sim_Timer(IN := FALSE);
    END_IF;
    
    Discharge_Active := FALSE;
    IF Step >= 1 AND Step <= 10 THEN
        Discharge_Active := semi_auto_bin_motor[Step];
    END_IF;
    
    IF Discharge_Active THEN
        Sim_Timer(IN := TRUE, PT := T#1000S);
        load_cell_value := Start_Sim_Weight + (TIME_TO_REAL(Sim_Timer.ET) / 1000.0) * Sim_Rate;
    ELSE
        Sim_Timer(IN := FALSE);
        Start_Sim_Weight := load_cell_value;
    END_IF;
END_IF;

(* 4. RECIPE SEQUENCE START & CYCLIC RESET *)
IF Step = 0 AND Start_Button THEN
    Step := 1;
    bin_last_weight := load_cell_value; (* Snapshot relative tare at whatever weight scale is *)
    Sequence_Complete := FALSE;
    Excess_Alarm := FALSE;
    Error_Code := 0;
    Status_Message := 'Semi-Auto Pour Started';
    Active_Target_Weight := 0.0;
    Active_Live_Weight := 0.0;
    FOR i := 1 TO 10 DO
        Actual_Weights[i] := 0.0;
        Semi_Auto_Bin[i] := FALSE;
        semi_auto_bin_cutoff[i] := FALSE;
        semi_auto_bin_motor[i] := FALSE;
    END_FOR;
END_IF;

(* 5. SEQUENCE CONTROL STATE MACHINE *)
CASE Step OF
    0:
        Active_Material_ID := 0;
        Active_Bin_ID := 0;
        Active_Target_Weight := 0.0;
        Active_Live_Weight := 0.0;
        Excess_Alarm := FALSE;
        Sequence_Complete := FALSE;
        FOR i := 1 TO 10 DO
            Semi_Auto_Bin[i] := FALSE;
            semi_auto_bin_cutoff[i] := FALSE;
            semi_auto_bin_motor[i] := FALSE;
        END_FOR;
        IF Error_Code = 0 THEN Status_Message := 'Semi-Auto Idle'; END_IF;
        
    1..10: (* DISCHARGE SILOS 1 TO 10 *)
        Mat_Idx := Semi_Auto_Bin_Material_Mapping[Step];
        
        (* Skip this step instantly if material mapping is 0 OR target weight is 0.0 kg *)
        IF Mat_Idx = 0 OR (Mat_Idx <= 20 AND GVL.Recipe_Weights[Mat_Idx] = 0.0) THEN
            IF Step = 10 THEN
                Step := 31; (* Transition directly to final settling delay *)
            ELSE
                Step := Step + 1;
            END_IF;
        ELSE
            target_weight := GVL.Recipe_Weights[Mat_Idx];
            cutoff_trigger_weight := target_weight - Semi_Auto_Coarse_To_Fine_speed[Step];
            min_tol_weight := target_weight - Semi_Auto_Bin_Tolerance[Step];
            max_tol_weight := target_weight + Semi_Auto_Bin_Tolerance[Step];
            
            Active_Target_Weight := target_weight;
            actual_bin := load_cell_value - bin_last_weight;
            Actual_Weights[Step] := actual_bin;
            Active_Live_Weight := actual_bin; (* Live tared weight of active bin *)
            
            Active_Material_ID := Mat_Idx;
            Active_Bin_ID := Step; (* Direct 1..10 *)
            
            (* Scale Overload Protection *)
            IF load_cell_value > 500.0 THEN
                Error_Code := 21;
                Status_Message := 'Error 21: Scale Overloaded!';
                Sequence_Complete := TRUE;
                Paused_By_EStop := TRUE;
            END_IF;
            
            (* Real-Time Feed & Instant Excess Alarm *)
            IF actual_bin < cutoff_trigger_weight THEN
                (* Coarse Feed *)
                Semi_Auto_Bin[Step] := TRUE;
                semi_auto_bin_cutoff[Step] := FALSE;
                semi_auto_bin_motor[Step] := TRUE;
                Excess_Alarm := FALSE;
                Status_Message := 'Semi-Auto Pouring (Coarse Feed)';
                
            ELSIF actual_bin < min_tol_weight THEN
                (* Fine Feed *)
                Semi_Auto_Bin[Step] := FALSE;
                semi_auto_bin_cutoff[Step] := TRUE;
                semi_auto_bin_motor[Step] := TRUE;
                Excess_Alarm := FALSE;
                Status_Message := 'Semi-Auto Pouring (Fine Feed)';
                
            ELSIF actual_bin > max_tol_weight THEN
                (* Excess Weight -> Instant Alarm, No Delay! *)
                Semi_Auto_Bin[Step] := FALSE;
                semi_auto_bin_cutoff[Step] := FALSE;
                semi_auto_bin_motor[Step] := FALSE;
                
                IF Excess_Allowed THEN
                    Excess_Alarm := FALSE;
                    Status_Message := 'Excess Weight Allowed: Advancing';
                    bin_last_weight := load_cell_value;
                    Active_Target_Weight := 0.0;
                    Active_Live_Weight := 0.0;
                    IF Step = 10 THEN
                        Step := 31;
                    ELSE
                        Step := Step + 1;
                    END_IF;
                ELSE
                    Excess_Alarm := TRUE; (* Immediate Trigger! *)
                    Status_Message := 'Excess Alarm: Weight above max tolerance! Reduce weight.';
                END_IF;
                
            ELSE
                (* In Tolerance Window [Min_Tol .. Max_Tol] *)
                Semi_Auto_Bin[Step] := FALSE;
                semi_auto_bin_cutoff[Step] := FALSE;
                semi_auto_bin_motor[Step] := FALSE;
                Excess_Alarm := FALSE;
                bin_last_weight := load_cell_value;
                Active_Target_Weight := 0.0;
                Active_Live_Weight := 0.0;
                
                IF Step = 10 THEN
                    Step := 31;
                ELSE
                    Step := Step + 1;
                END_IF;
            END_IF;
        END_IF;

    31: (* POST-SEQUENCE FINAL SETTLING DELAY *)
        Active_Material_ID := 0;
        Active_Bin_ID := 0;
        Active_Target_Weight := 0.0;
        Active_Live_Weight := 0.0;
        Excess_Alarm := FALSE;
        Status_Message := 'Final Settling Delay';
        Completion_Timer(IN := TRUE, PT := Effective_Delay);
        IF Completion_Timer.Q THEN
            Completion_Timer(IN := FALSE);
            Step := 32;
        END_IF;
        
    32: (* COMPLETE *)
        Active_Material_ID := 0;
        Active_Bin_ID := 0;
        Active_Target_Weight := 0.0;
        Active_Live_Weight := 0.0;
        Excess_Alarm := FALSE;
        Status_Message := 'Sequence Completed';
        Sequence_Complete := TRUE;
        
        IF NOT Start_Button THEN
            Step := 0;
            Sequence_Complete := FALSE;
            FOR i := 1 TO 10 DO
                Actual_Weights[i] := 0.0;
            END_FOR;
        END_IF;
END_CASE;

END_FUNCTION_BLOCK

// PLC_AC500_V3/Application/old_version/batching13
PROGRAM batching13
VAR
    Auto_Ctrl : Auto_Batching_V13;
    Semi_Auto_Ctrl : Semi_Auto_Batching_V13;
    
    (* Sub-Block Diagnostic Indicators *)
    Auto_Err : INT;
    Auto_Msg : STRING;
    
    Semi_Auto_Err : INT;
    Semi_Auto_Msg : STRING;
    
    Auto_Complete : BOOL;
    Semi_Auto_Complete : BOOL;
    
    (* Repetitive Cycle Status *)
    Completed_Batch_Cycles : INT;      // Total completed batch cycle loops
    All_Cycles_Complete : BOOL;         // Indicator for full set completion
    
    (* Diagnostics & Interlocks *)
    Status_Message : STRING;
    
    i : INT;
    j : INT;
    Duplicate_Found : BOOL;
    Invalid_Material_Range : BOOL;
    Weight_Limit_Error : BOOL;
    
    (* Cycle Manager state variables *)
    Cycle_Manager_State : INT;         // State index for loop management
    Internal_FB_Start : BOOL;          // Controlled command to restart sub-blocks
END_VAR

(* 1. STARTUP CONFIGURATION, RECIPE TOTALS, AND WEIGHT CHECKS *)
Duplicate_Found := FALSE;
Invalid_Material_Range := FALSE;
Weight_Limit_Error := FALSE;

(* Calculate Auto Total Target Weight & Material Count *)
GVL.Auto_Total_Target_Weight := 0.0;
GVL.Auto_Material_Count := 0;
FOR i := 1 TO 6 DO
    (* Check 2: Out of Range (Auto) *)
    IF GVL.Auto_Bin_Material_Mapping[i] < 0 OR GVL.Auto_Bin_Material_Mapping[i] > 20 THEN
        Invalid_Material_Range := TRUE;
    END_IF;
    
    (* Check 1: Duplicate Cross-Array Material ID *)
    IF GVL.Auto_Bin_Material_Mapping[i] <> 0 AND GVL.Auto_Bin_Material_Mapping[i] <= 20 THEN
        FOR j := 1 TO 10 DO
            IF GVL.Auto_Bin_Material_Mapping[i] = GVL.Semi_Auto_Bin_Material_Mapping[j] THEN
                Duplicate_Found := TRUE;
            END_IF;
        END_FOR;
    END_IF;
    
    (* Accumulate Auto Total Target Weight and Active Count *)
    IF GVL.Auto_Bin_Material_Mapping[i] > 0 AND GVL.Auto_Bin_Material_Mapping[i] <= 20 THEN
        IF GVL.Recipe_Weights[GVL.Auto_Bin_Material_Mapping[i]] > 0.0 THEN
            GVL.Auto_Total_Target_Weight := GVL.Auto_Total_Target_Weight + GVL.Recipe_Weights[GVL.Auto_Bin_Material_Mapping[i]];
            GVL.Auto_Material_Count := GVL.Auto_Material_Count + 1;
            
            (* Check 3: Recipe weight is less than Cutoff + Tolerance *)
            IF GVL.Recipe_Weights[GVL.Auto_Bin_Material_Mapping[i]] < (GVL.Auto_Coarse_To_Fine_speed[i] + GVL.Auto_Bin_Tolerance[i]) THEN
                Weight_Limit_Error := TRUE;
            END_IF;
        END_IF;
    END_IF;
END_FOR;

(* Calculate Semi-Auto Total Target Weight & Material Count *)
GVL.Semi_Auto_Total_Target_Weight := 0.0;
GVL.Semi_Auto_Material_Count := 0;
FOR j := 1 TO 10 DO
    (* Check 2: Out of Range (Semi-Auto) *)
    IF GVL.Semi_Auto_Bin_Material_Mapping[j] < 0 OR GVL.Semi_Auto_Bin_Material_Mapping[j] > 20 THEN
        Invalid_Material_Range := TRUE;
    END_IF;
    
    (* Accumulate Semi-Auto Total Target Weight and Active Count *)
    IF GVL.Semi_Auto_Bin_Material_Mapping[j] > 0 AND GVL.Semi_Auto_Bin_Material_Mapping[j] <= 20 THEN
        IF GVL.Recipe_Weights[GVL.Semi_Auto_Bin_Material_Mapping[j]] > 0.0 THEN
            GVL.Semi_Auto_Total_Target_Weight := GVL.Semi_Auto_Total_Target_Weight + GVL.Recipe_Weights[GVL.Semi_Auto_Bin_Material_Mapping[j]];
            GVL.Semi_Auto_Material_Count := GVL.Semi_Auto_Material_Count + 1;
            
            (* Check 3: Recipe weight check (Semi-Auto) *)
            IF GVL.Recipe_Weights[GVL.Semi_Auto_Bin_Material_Mapping[j]] < (GVL.Semi_Auto_Coarse_To_Fine_speed[j] + GVL.Semi_Auto_Bin_Tolerance[j]) THEN
                Weight_Limit_Error := TRUE;
            END_IF;
        END_IF;
    END_IF;
END_FOR;

(* Configuration Error Resolution *)
IF Duplicate_Found THEN
    GVL.Error_Code := 1;
    Status_Message := 'Error 1: Duplicate Material ID mapped in Auto and Semi-Auto!';
ELSIF Invalid_Material_Range THEN
    GVL.Error_Code := 2;
    Status_Message := 'Error 2: Material Index configuration out of range (1..20)!';
ELSIF Weight_Limit_Error THEN
    GVL.Error_Code := 3;
    Status_Message := 'Error 3: Recipe weight is less than Cutoff + Tolerance!';
ELSE
    IF GVL.Error_Code <= 3 THEN
        GVL.Error_Code := 0;
    END_IF;
END_IF;

(* Abort / Hard Reset Interlock *)
IF (GVL.Error_Code >= 1 AND GVL.Error_Code <= 3) OR GVL.Reset THEN
    FOR i := 1 TO 6 DO 
        GVL.Auto_Bin[i] := FALSE; 
        GVL.auto_bin_cutoff[i] := FALSE; 
        GVL.auto_bin_motor[i] := FALSE; 
        GVL.Auto_Weights[i] := 0.0;
    END_FOR;
    
    FOR i := 1 TO 10 DO 
        GVL.Semi_Auto_Bin[i] := FALSE; 
        GVL.semi_auto_bin_cutoff[i] := FALSE; 
        GVL.semi_auto_bin_motor[i] := FALSE; 
        GVL.Semi_Auto_Weights[i] := 0.0;
    END_FOR;
    
    Internal_FB_Start := FALSE;
    Auto_Ctrl(Start_Button := FALSE, E_Stop_Active := FALSE, Reset := GVL.Reset, load_cell_value := GVL.load_cell_auto, Inter_Bin_Delay := GVL.Auto_Inter_Bin_Delay, Excess_Allowed := GVL.Auto_Excess_Allowed);
    Semi_Auto_Ctrl(Start_Button := FALSE, E_Stop_Active := FALSE, Reset := GVL.Reset, load_cell_value := GVL.load_cell_semi_auto, Inter_Bin_Delay := GVL.Semi_Auto_Inter_Bin_Delay, Excess_Allowed := GVL.Semi_Auto_Excess_Allowed);
    
    GVL.Auto_Active_Target_Weight := 0.0;
    GVL.Auto_Active_Live_Weight := 0.0;
    GVL.Semi_Auto_Active_Target_Weight := 0.0;
    GVL.Semi_Auto_Active_Live_Weight := 0.0;
    
    Auto_Complete := TRUE;
    Semi_Auto_Complete := TRUE;
    All_Cycles_Complete := TRUE;
    
    GVL.Cycle_Hold_Active := FALSE;
    GVL.Run := FALSE;
    Cycle_Manager_State := 0;
    
    IF GVL.Reset THEN
        GVL.Error_Code := 0;
        GVL.Current_Batch_Cycle := 0;
        GVL.Target_Batch_Cycles := 0;
        GVL.Start_Button := FALSE;
        Completed_Batch_Cycles := 0;
        Status_Message := 'System Reset Activated';
        Auto_Complete := FALSE;
        Semi_Auto_Complete := FALSE;
        All_Cycles_Complete := FALSE;
        
        GVL.Auto_Active_Mat := 0;
        GVL.Auto_Active_Bin := 0;
        GVL.Semi_Auto_Active_Mat := 0;
        GVL.Semi_Auto_Active_Bin := 0;
        GVL.Auto_Excess_Alarm := FALSE;
        GVL.Semi_Auto_Excess_Alarm := FALSE;
        
        (* Auto-clearing trigger: set Reset back to FALSE *)
        GVL.Reset := FALSE;
    END_IF;
    RETURN;
END_IF;


(* 2. REPETITIVE CYCLE MANAGER STATE MACHINE WITH PRE-RUN INITIAL TOLERANCE CHECK *)
CASE Cycle_Manager_State OF
    0: (* IDLE STATE *)
        Internal_FB_Start := FALSE;
        All_Cycles_Complete := FALSE;
        GVL.Cycle_Hold_Active := FALSE;
        GVL.Run := FALSE;
        IF GVL.Error_Code = 0 AND Status_Message <> 'Error: Target Batch Cycles is 0!' AND Status_Message <> 'Error 4: Scale weight exceeds Initial Tolerance!' THEN 
            Status_Message := 'System Ready'; 
        END_IF;
        
